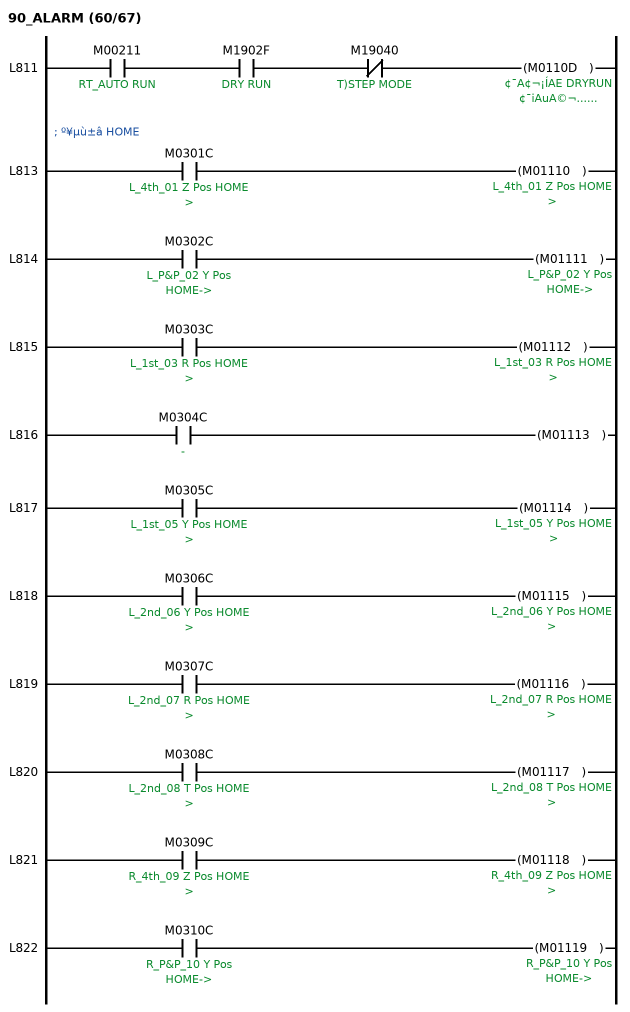
[picture p456: 90_ALARM rungs L811-L822]
; L811
LOAD      M00211	// RT_AUTO RUN
AND       M1902F	// DRY RUN
AND NOT   M19040	// T)STEP MODE
OUT       M0110D	// ¢¯A¢¬¡ÍAE DRYRUN ¢¯iAuA©¬......
// º¥µù±â HOME
; L813
LOAD      M0301C	// L_4th_01 Z Pos HOME >
OUT       M01110	// L_4th_01 Z Pos HOME >
; L814
LOAD      M0302C	// L_P&P_02 Y Pos HOME->
OUT       M01111	// L_P&P_02 Y Pos HOME->
; L815
LOAD      M0303C	// L_1st_03 R Pos HOME >
OUT       M01112	// L_1st_03 R Pos HOME >
; L816
LOAD      M0304C	// -
OUT       M01113
; L817
LOAD      M0305C	// L_1st_05 Y Pos HOME >
OUT       M01114	// L_1st_05 Y Pos HOME >
; L818
LOAD      M0306C	// L_2nd_06 Y Pos HOME >
OUT       M01115	// L_2nd_06 Y Pos HOME >
; L819
LOAD      M0307C	// L_2nd_07 R Pos HOME >
OUT       M01116	// L_2nd_07 R Pos HOME >
; L820
LOAD      M0308C	// L_2nd_08 T Pos HOME >
OUT       M01117	// L_2nd_08 T Pos HOME >
; L821
LOAD      M0309C	// R_4th_09 Z Pos HOME >
OUT       M01118	// R_4th_09 Z Pos HOME >
; L822
LOAD      M0310C	// R_P&P_10 Y Pos HOME->
OUT       M01119	// R_P&P_10 Y Pos HOME->

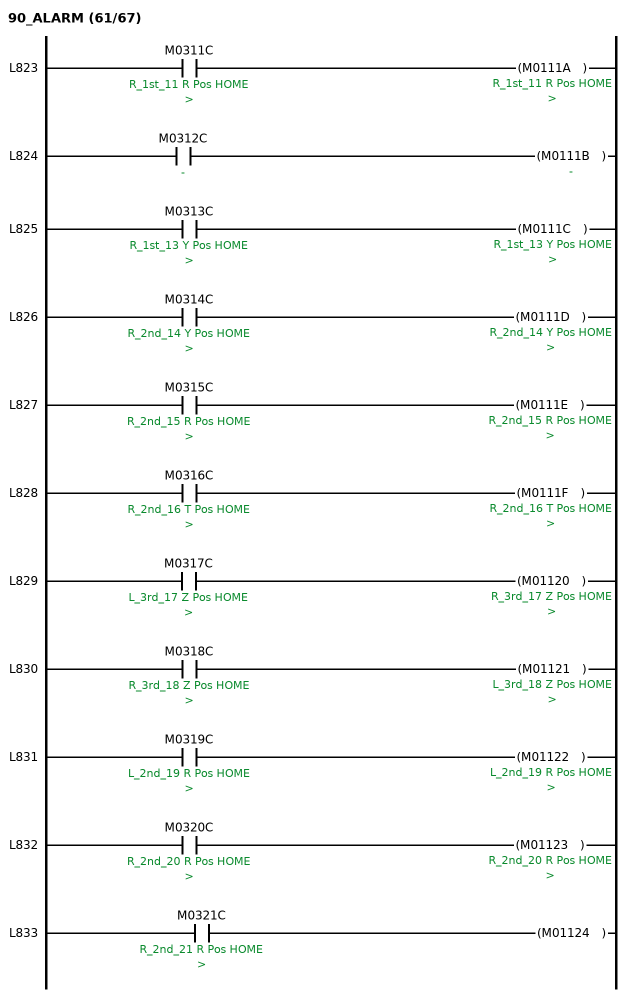
; L823
LOAD      M0311C	// R_1st_11 R Pos HOME >
OUT       M0111A	// R_1st_11 R Pos HOME >
; L824
LOAD      M0312C	// -
OUT       M0111B	// -
; L825
LOAD      M0313C	// R_1st_13 Y Pos HOME >
OUT       M0111C	// R_1st_13 Y Pos HOME >
; L826
LOAD      M0314C	// R_2nd_14 Y Pos HOME >
OUT       M0111D	// R_2nd_14 Y Pos HOME >
; L827
LOAD      M0315C	// R_2nd_15 R Pos HOME >
OUT       M0111E	// R_2nd_15 R Pos HOME >
; L828
LOAD      M0316C	// R_2nd_16 T Pos HOME >
OUT       M0111F	// R_2nd_16 T Pos HOME >
; L829
LOAD      M0317C	// L_3rd_17 Z Pos HOME >
OUT       M01120	// R_3rd_17 Z Pos HOME >
; L830
LOAD      M0318C	// R_3rd_18 Z Pos HOME >
OUT       M01121	// L_3rd_18 Z Pos HOME >
; L831
LOAD      M0319C	// L_2nd_19 R Pos HOME >
OUT       M01122	// L_2nd_19 R Pos HOME >
; L832
LOAD      M0320C	// R_2nd_20 R Pos HOME >
OUT       M01123	// R_2nd_20 R Pos HOME >
; L833
LOAD      M0321C	// R_2nd_21 R Pos HOME >
OUT       M01124

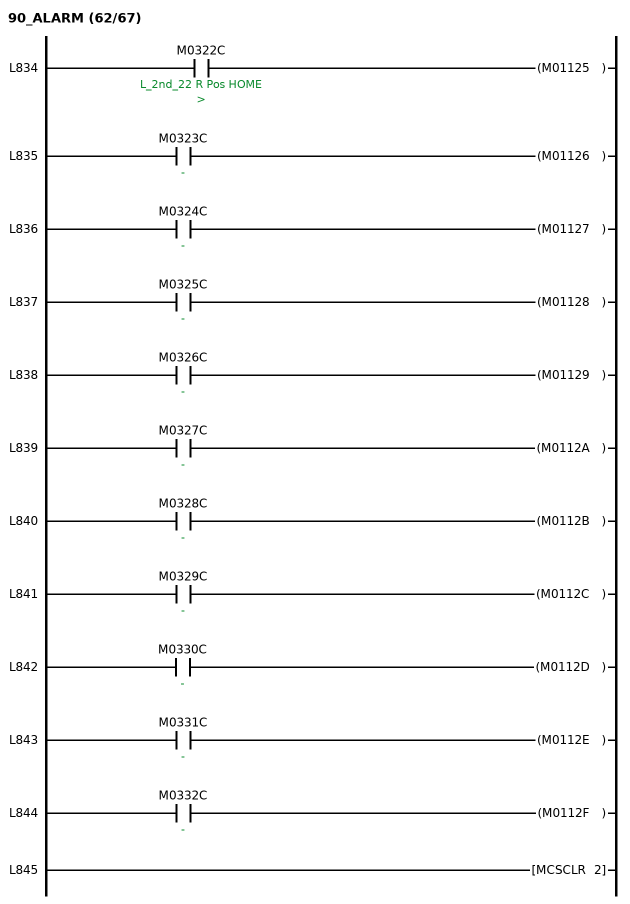
; L834
LOAD      M0322C	// L_2nd_22 R Pos HOME >
OUT       M01125
; L835
LOAD      M0323C	// -
OUT       M01126
; L836
LOAD      M0324C	// -
OUT       M01127
; L837
LOAD      M0325C	// -
OUT       M01128
; L838
LOAD      M0326C	// -
OUT       M01129
; L839
LOAD      M0327C	// -
OUT       M0112A
; L840
LOAD      M0328C	// -
OUT       M0112B
; L841
LOAD      M0329C	// -
OUT       M0112C
; L842
LOAD      M0330C	// -
OUT       M0112D
; L843
LOAD      M0331C	// -
OUT       M0112E
; L844
LOAD      M0332C	// -
OUT       M0112F
; L845
MCSCLR    2

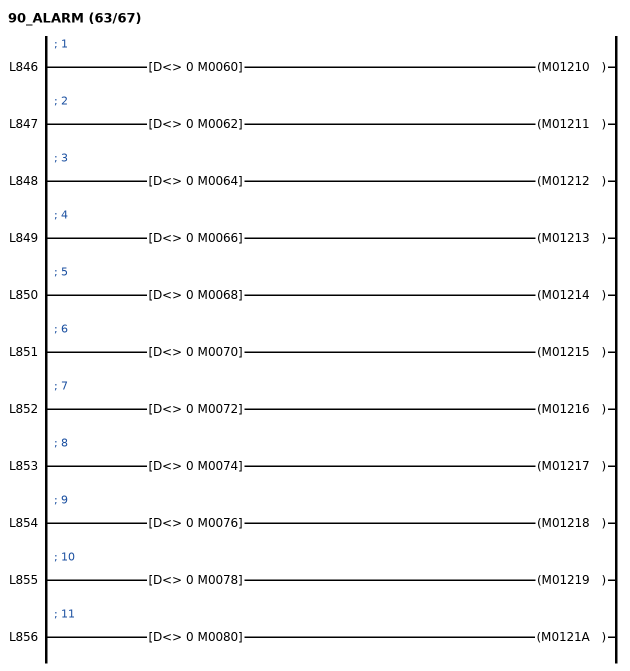
; L846
LOADD<>   0 M0060
OUT       M01210
// output comment: 1
; L847
LOADD<>   0 M0062
OUT       M01211
// output comment: 2
; L848
LOADD<>   0 M0064
OUT       M01212
// output comment: 3
; L849
LOADD<>   0 M0066
OUT       M01213
// output comment: 4
; L850
LOADD<>   0 M0068
OUT       M01214
// output comment: 5
; L851
LOADD<>   0 M0070
OUT       M01215
// output comment: 6
; L852
LOADD<>   0 M0072
OUT       M01216
// output comment: 7
; L853
LOADD<>   0 M0074
OUT       M01217
// output comment: 8
; L854
LOADD<>   0 M0076
OUT       M01218
// output comment: 9
; L855
LOADD<>   0 M0078
OUT       M01219
// output comment: 10
; L856
LOADD<>   0 M0080
OUT       M0121A
// output comment: 11

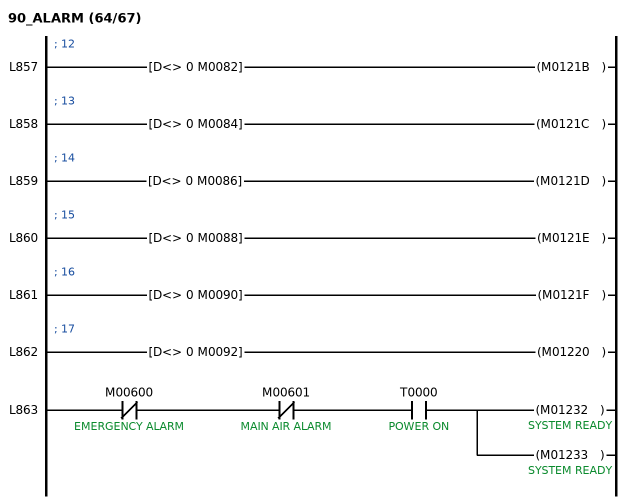
; L857
LOADD<>   0 M0082
OUT       M0121B
// output comment: 12
; L858
LOADD<>   0 M0084
OUT       M0121C
// output comment: 13
; L859
LOADD<>   0 M0086
OUT       M0121D
// output comment: 14
; L860
LOADD<>   0 M0088
OUT       M0121E
// output comment: 15
; L861
LOADD<>   0 M0090
OUT       M0121F
// output comment: 16
; L862
LOADD<>   0 M0092
OUT       M01220
// output comment: 17
; L863
LOAD NOT  M00600	// EMERGENCY ALARM
AND NOT   M00601	// MAIN AIR ALARM
AND       T0000	// POWER ON
OUT       M01232	// SYSTEM READY
OUT       M01233	// SYSTEM READY

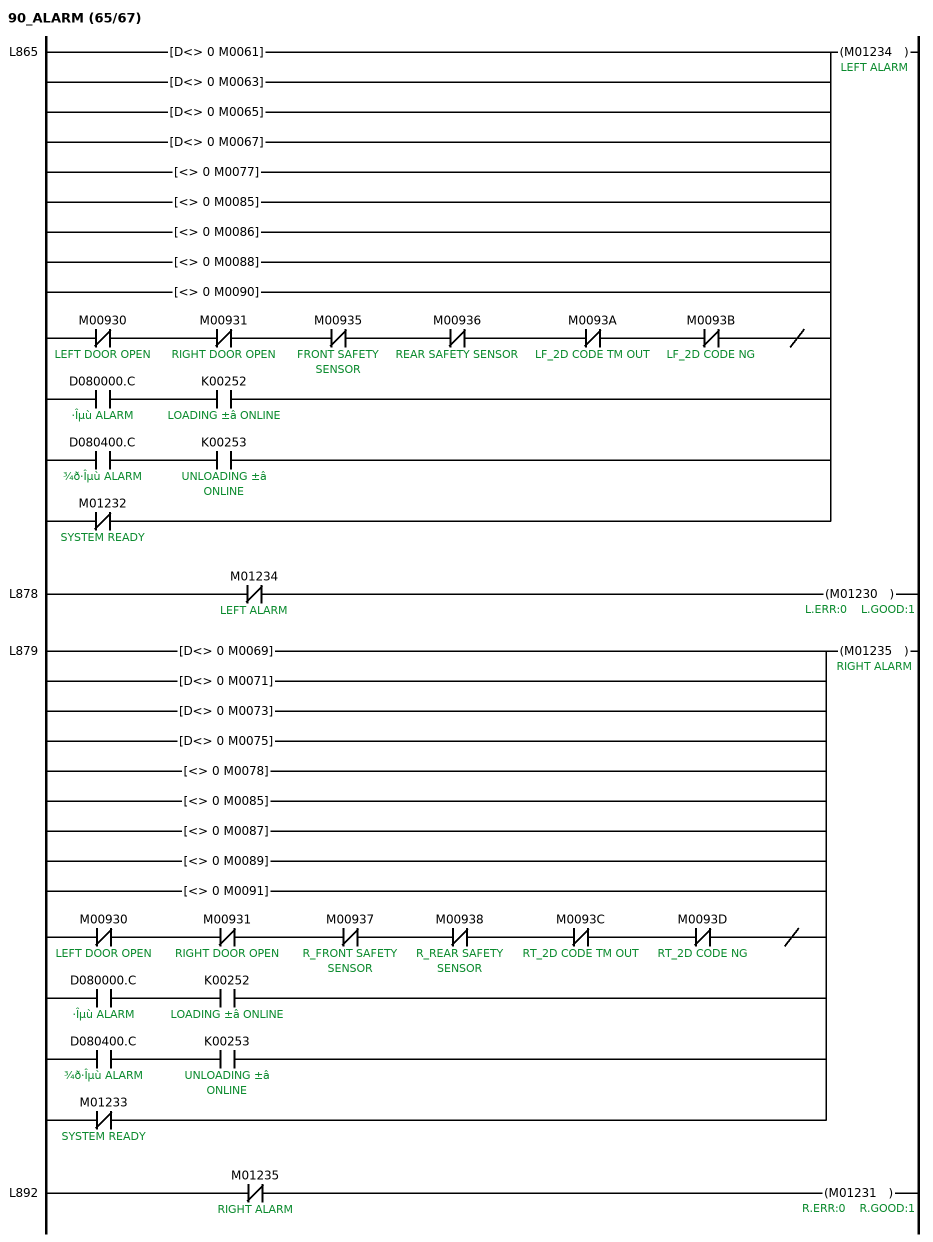
; L865
LOADD<>   0 M0061
ORD<>     0 M0063
ORD<>     0 M0065
ORD<>     0 M0067
OR<>      0 M0077
OR<>      0 M0085
OR<>      0 M0086
OR<>      0 M0088
OR<>      0 M0090
LOAD NOT  M00930	// LEFT DOOR OPEN
AND NOT   M00931	// RIGHT DOOR OPEN
AND NOT   M00935	// FRONT SAFETY SENSOR
AND NOT   M00936	// REAR SAFETY SENSOR
AND NOT   M0093A	// LF_2D CODE TM OUT
AND NOT   M0093B	// LF_2D CODE NG
NOT
OR LOAD
LOAD      D080000.C	// ·Îµù ALARM
AND       K00252	// LOADING ±â ONLINE
OR LOAD
LOAD      D080400.C	// ¾ð·Îµù ALARM
AND       K00253	// UNLOADING ±â ONLINE
OR LOAD
OR NOT    M01232	// SYSTEM READY
OUT       M01234	// LEFT ALARM
; L878
LOAD NOT  M01234	// LEFT ALARM
OUT       M01230	// L.ERR:0    L.GOOD:1
; L879
LOADD<>   0 M0069
ORD<>     0 M0071
ORD<>     0 M0073
ORD<>     0 M0075
OR<>      0 M0078
OR<>      0 M0085
OR<>      0 M0087
OR<>      0 M0089
OR<>      0 M0091
LOAD NOT  M00930	// LEFT DOOR OPEN
AND NOT   M00931	// RIGHT DOOR OPEN
AND NOT   M00937	// R_FRONT SAFETY SENSOR
AND NOT   M00938	// R_REAR SAFETY SENSOR
AND NOT   M0093C	// RT_2D CODE TM OUT
AND NOT   M0093D	// RT_2D CODE NG
NOT
OR LOAD
LOAD      D080000.C	// ·Îµù ALARM
AND       K00252	// LOADING ±â ONLINE
OR LOAD
LOAD      D080400.C	// ¾ð·Îµù ALARM
AND       K00253	// UNLOADING ±â ONLINE
OR LOAD
OR NOT    M01233	// SYSTEM READY
OUT       M01235	// RIGHT ALARM
; L892
LOAD NOT  M01235	// RIGHT ALARM
OUT       M01231	// R.ERR:0    R.GOOD:1

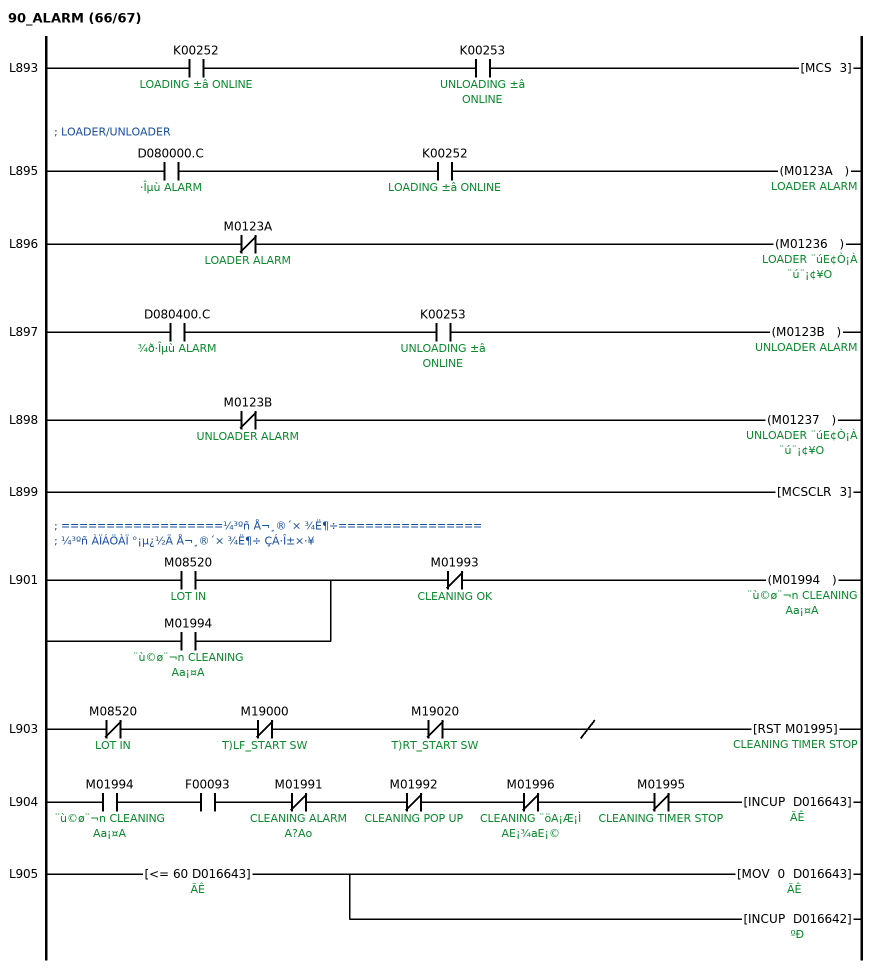
; L893
LOAD      K00252	// LOADING ±â ONLINE
AND       K00253	// UNLOADING ±â ONLINE
MCS       3
// LOADER/UNLOADER
; L895
LOAD      D080000.C	// ·Îµù ALARM
AND       K00252	// LOADING ±â ONLINE
OUT       M0123A	// LOADER ALARM
; L896
LOAD NOT  M0123A	// LOADER ALARM
OUT       M01236	// LOADER ¨úE¢Ò¡À ¨ú¨¡¢¥O
; L897
LOAD      D080400.C	// ¾ð·Îµù ALARM
AND       K00253	// UNLOADING ±â ONLINE
OUT       M0123B	// UNLOADER ALARM
; L898
LOAD NOT  M0123B	// UNLOADER ALARM
OUT       M01237	// UNLOADER ¨úE¢Ò¡À ¨ú¨¡¢¥O
; L899
MCSCLR    3
// ==================¼³ºñ Å¬¸®´× ¾Ë¶÷================
; L901
LOAD      M08520	// LOT IN
OR        M01994	// ¨ù©ø¨¬n CLEANING Aa¡¤A
AND NOT   M01993	// CLEANING OK
OUT       M01994	// ¨ù©ø¨¬n CLEANING Aa¡¤A
// output comment: ¼³ºñ ÀÏÁÖÀÏ °¡µ¿½Ã Å¬¸®´× ¾Ë¶÷ ÇÁ·Î±×·¥
; L903
LOAD NOT  M08520	// LOT IN
AND NOT   M19000	// T)LF_START SW
AND NOT   M19020	// T)RT_START SW
NOT
RST       M01995	// CLEANING TIMER STOP
; L904
LOAD      M01994	// ¨ù©ø¨¬n CLEANING Aa¡¤A
AND       F00093
AND NOT   M01991	// CLEANING ALARM A?Ao
AND NOT   M01992	// CLEANING POP UP
AND NOT   M01996	// CLEANING ¨öA¡Æ¡Ì AE¡¾aE¡©
AND NOT   M01995	// CLEANING TIMER STOP
INCUP     D016643	// ÃÊ
; L905
LOAD<=    60 D016643	// ÃÊ
MOV       0 D016643	// ÃÊ
INCUP     D016642	// ºÐ

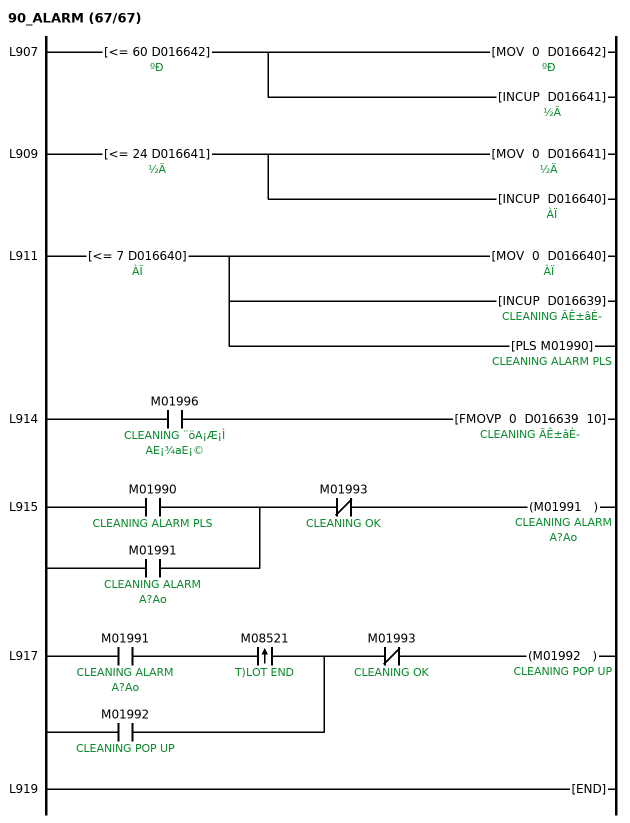
; L907
LOAD<=    60 D016642	// ºÐ
MOV       0 D016642	// ºÐ
INCUP     D016641	// ½Ã
; L909
LOAD<=    24 D016641	// ½Ã
MOV       0 D016641	// ½Ã
INCUP     D016640	// ÀÏ
; L911
LOAD<=    7 D016640	// ÀÏ
MOV       0 D016640	// ÀÏ
INCUP     D016639	// CLEANING ÃÊ±âÈ­
OUTP      M01990	// CLEANING ALARM PLS
; L914
LOAD      M01996	// CLEANING ¨öA¡Æ¡Ì AE¡¾aE¡©
FMOVP     0 D016639 10	// CLEANING ÃÊ±âÈ­
; L915
LOAD      M01990	// CLEANING ALARM PLS
OR        M01991	// CLEANING ALARM A?Ao
AND NOT   M01993	// CLEANING OK
OUT       M01991	// CLEANING ALARM A?Ao
; L917
LOAD      M01991	// CLEANING ALARM A?Ao
ANDP      M08521	// T)LOT END
OR        M01992	// CLEANING POP UP
AND NOT   M01993	// CLEANING OK
OUT       M01992	// CLEANING POP UP
; L919
END

PROGRAM 91_DEVICE_CHANGE (task: ½ºÄµ ÇÁ·Î±×·¥)

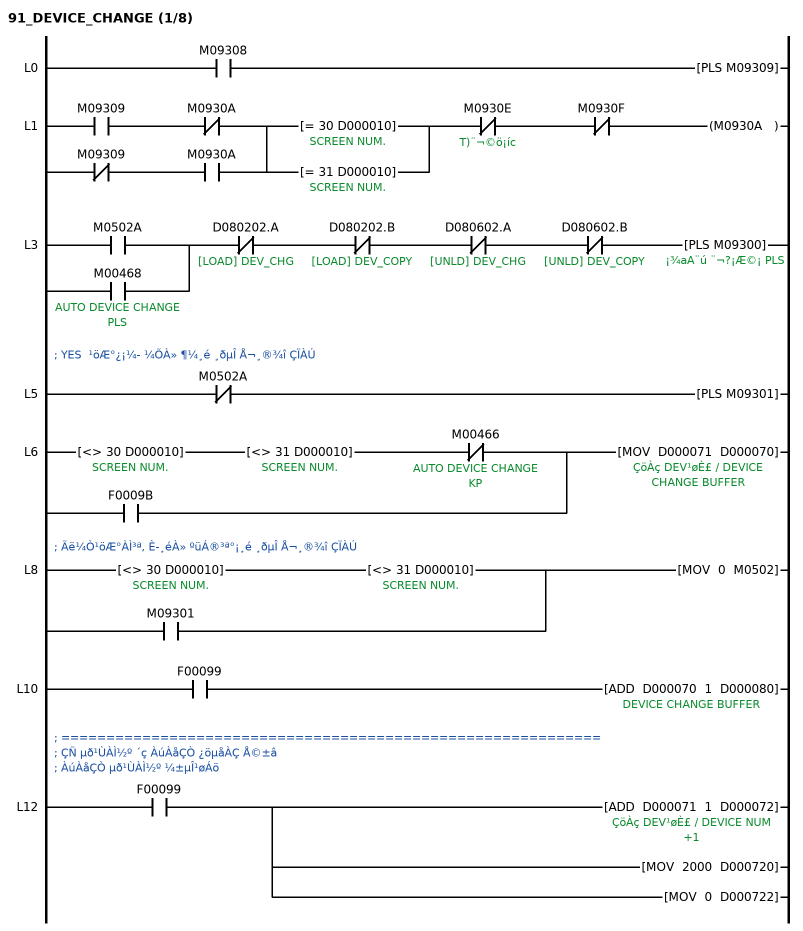
; L0
LOAD      M09308
OUTP      M09309
; L1
LOAD      M09309
AND NOT   M0930A
LOAD NOT  M09309
AND       M0930A
OR LOAD
LOAD=     30 D000010	// SCREEN NUM.
OR=       31 D000010	// SCREEN NUM.
AND LOAD
AND NOT   M0930E	// T)¨¬©ö¡íc
AND NOT   M0930F
OUT       M0930A
; L3
LOAD      M0502A
OR        M00468	// AUTO DEVICE CHANGE PLS
AND NOT   D080202.A	// [LOAD] DEV_CHG
AND NOT   D080202.B	// [LOAD] DEV_COPY
AND NOT   D080602.A	// [UNLD] DEV_CHG
AND NOT   D080602.B	// [UNLD] DEV_COPY
OUTP      M09300	// ¡¾aA¨ú ¨¬?¡Æ©¡ PLS
; L5
LOAD NOT  M0502A
OUTP      M09301
// output comment: YES  ¹öÆ°¿¡¼­ ¼ÕÀ» ¶¼¸é ¸ðµÎ Å¬¸®¾î ÇÏÀÚ
; L6
LOAD<>    30 D000010	// SCREEN NUM.
AND<>     31 D000010	// SCREEN NUM.
AND NOT   M00466	// AUTO DEVICE CHANGE KP
OR        F0009B
MOV       D000071 D000070	// ÇöÀç DEV¹øÈ£ / DEVICE CHANGE BUFFER
; L8
LOAD<>    30 D000010	// SCREEN NUM.
AND<>     31 D000010	// SCREEN NUM.
OR        M09301
MOV       0 M0502
// output comment: Ãë¼Ò¹öÆ°ÀÌ³ª, È­¸éÀ» ºüÁ®³ª°¡¸é ¸ðµÎ Å¬¸®¾î ÇÏÀÚ
; L10
LOAD      F00099
ADD       D000070 1 D000080	// DEVICE CHANGE BUFFER
// ============================================================
; L12
LOAD      F00099
ADD       D000071 1 D000072	// ÇöÀç DEV¹øÈ£ / DEVICE NUM +1
MOV       2000 D000720
MOV       0 D000722
// output comment: ÇÑ µð¹ÙÀÌ½º ´ç ÀúÀåÇÒ ¿öµåÀÇ Å©±â
// output comment: ÀúÀåÇÒ µð¹ÙÀÌ½º ¼±µÎ¹øÁö

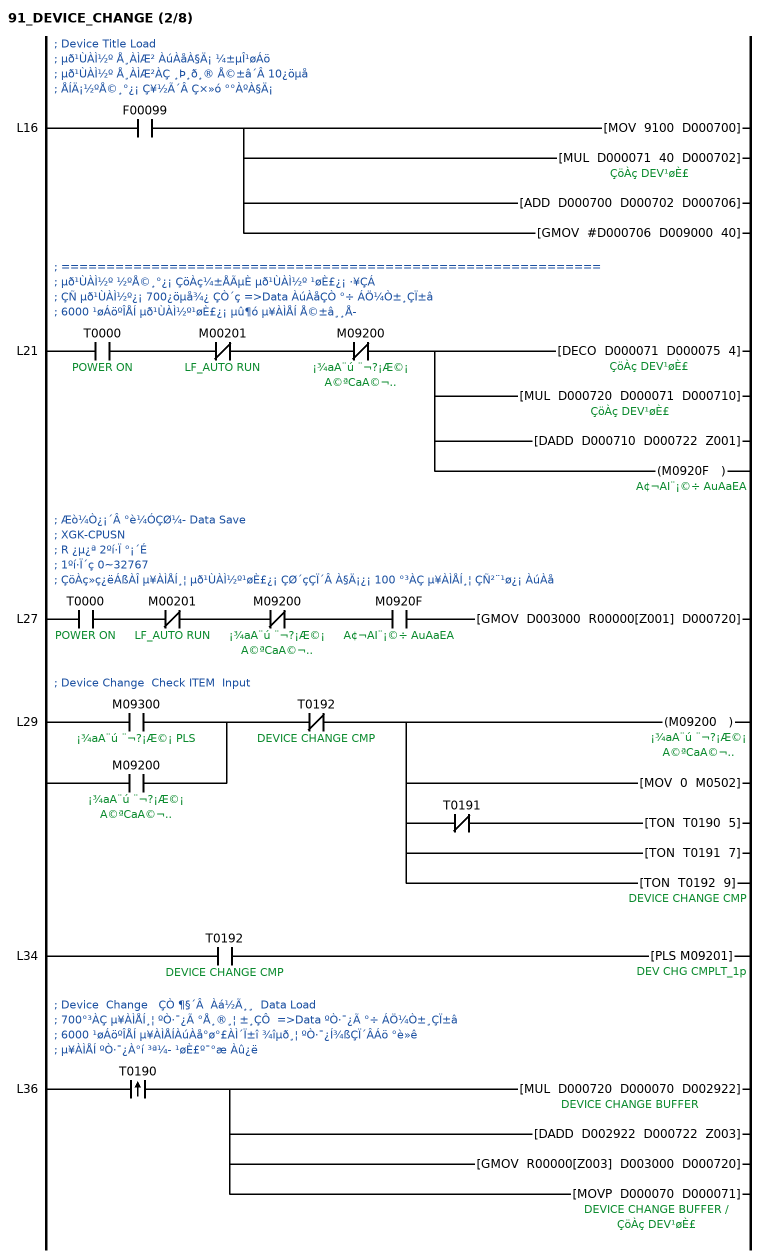
// Device Title Load
; L16
LOAD      F00099
MOV       9100 D000700
MUL       D000071 40 D000702	// ÇöÀç DEV¹øÈ£
ADD       D000700 D000702 D000706
GMOV      #D000706 D009000 40
// output comment: µð¹ÙÀÌ½º Å¸ÀÌÆ² ÀúÀåÀ§Ä¡ ¼±µÎ¹øÁö
// output comment: µð¹ÙÀÌ½º Å¸ÀÌÆ²ÀÇ ¸Þ¸ð¸® Å©±â´Â 10¿öµå
// output comment: ÅÍÄ¡½ºÅ©¸°¿¡ Ç¥½Ã´Â Ç×»ó °°ÀºÀ§Ä¡
// ============================================================
; L21
LOAD      T0000	// POWER ON
AND NOT   M00201	// LF_AUTO RUN
AND NOT   M09200	// ¡¾aA¨ú ¨¬?¡Æ©¡ A©ªCaA©¬..
DECO      D000071 D000075 4	// ÇöÀç DEV¹øÈ£
MUL       D000720 D000071 D000710	// ÇöÀç DEV¹øÈ£
DADD      D000710 D000722 Z001
OUT       M0920F	// A¢¬AI¨¡©÷ AuAaEA
// output comment: µð¹ÙÀÌ½º ½ºÅ©¸°¿¡ ÇöÀç¼±ÅÃµÈ µð¹ÙÀÌ½º ¹øÈ£¿¡ ·¥ÇÁ
// output comment: ÇÑ µð¹ÙÀÌ½º¿¡ 700¿öµå¾¿ ÇÒ´ç =>Data ÀúÀåÇÒ °÷ ÁÖ¼Ò±¸ÇÏ±â
// output comment: 6000 ¹øÁöºÎÅÍ µð¹ÙÀÌ½º¹øÈ£¿¡ µû¶ó µ¥ÀÌÅÍ Å©±â¸¸Å­
// Æò¼Ò¿¡´Â °è¼ÓÇØ¼­ Data Save
// XGK-CPUSN
// R ¿µ¿ª 2ºí·Ï °¡´É
// 1ºí·Ï´ç 0~32767
; L27
LOAD      T0000	// POWER ON
AND NOT   M00201	// LF_AUTO RUN
AND NOT   M09200	// ¡¾aA¨ú ¨¬?¡Æ©¡ A©ªCaA©¬..
AND       M0920F	// A¢¬AI¨¡©÷ AuAaEA
GMOV      D003000 R00000[Z001] D000720
// output comment: ÇöÀç»ç¿ëÁßÀÎ µ¥ÀÌÅÍ¸¦ µð¹ÙÀÌ½º¹øÈ£¿¡ ÇØ´çÇÏ´Â À§Ä¡¿¡ 100 °³ÀÇ µ¥ÀÌÅÍ¸¦ ÇÑ²¨¹ø¿¡ ÀúÀå
// Device Change  Check ITEM  Input
; L29
LOAD      M09300	// ¡¾aA¨ú ¨¬?¡Æ©¡ PLS
OR        M09200	// ¡¾aA¨ú ¨¬?¡Æ©¡ A©ªCaA©¬..
AND NOT   T0192	// DEVICE CHANGE CMP
OUT       M09200	// ¡¾aA¨ú ¨¬?¡Æ©¡ A©ªCaA©¬..
MOV       0 M0502
MPUSH
AND NOT   T0191
TON       T0190 5
MPOP
TON       T0191 7
TON       T0192 9	// DEVICE CHANGE CMP
; L34
LOAD      T0192	// DEVICE CHANGE CMP
OUTP      M09201	// DEV CHG CMPLT_1p
// Device  Change   ÇÒ ¶§´Â  Àá½Ã¸¸  Data Load
; L36
LOADP     T0190
MUL       D000720 D000070 D002922	// DEVICE CHANGE BUFFER
DADD      D002922 D000722 Z003
GMOV      R00000[Z003] D003000 D000720
MOVP      D000070 D000071	// DEVICE CHANGE BUFFER / ÇöÀç DEV¹øÈ£
// output comment: 700°³ÀÇ µ¥ÀÌÅÍ¸¦ ºÒ·¯¿Ã °Å¸®¸¦ ±¸ÇÔ  =>Data ºÒ·¯¿Ã °÷ ÁÖ¼Ò±¸ÇÏ±â
// output comment: 6000 ¹øÁöºÎÅÍ µ¥ÀÌÅÍÀúÀå°ø°£ÀÌ´Ï±î ¾îµð¸¦ ºÒ·¯¿Í¾ßÇÏ´ÂÁö °è»ê
// output comment: µ¥ÀÌÅÍ ºÒ·¯¿À°í ³ª¼­ ¹øÈ£º¯°æ Àû¿ë

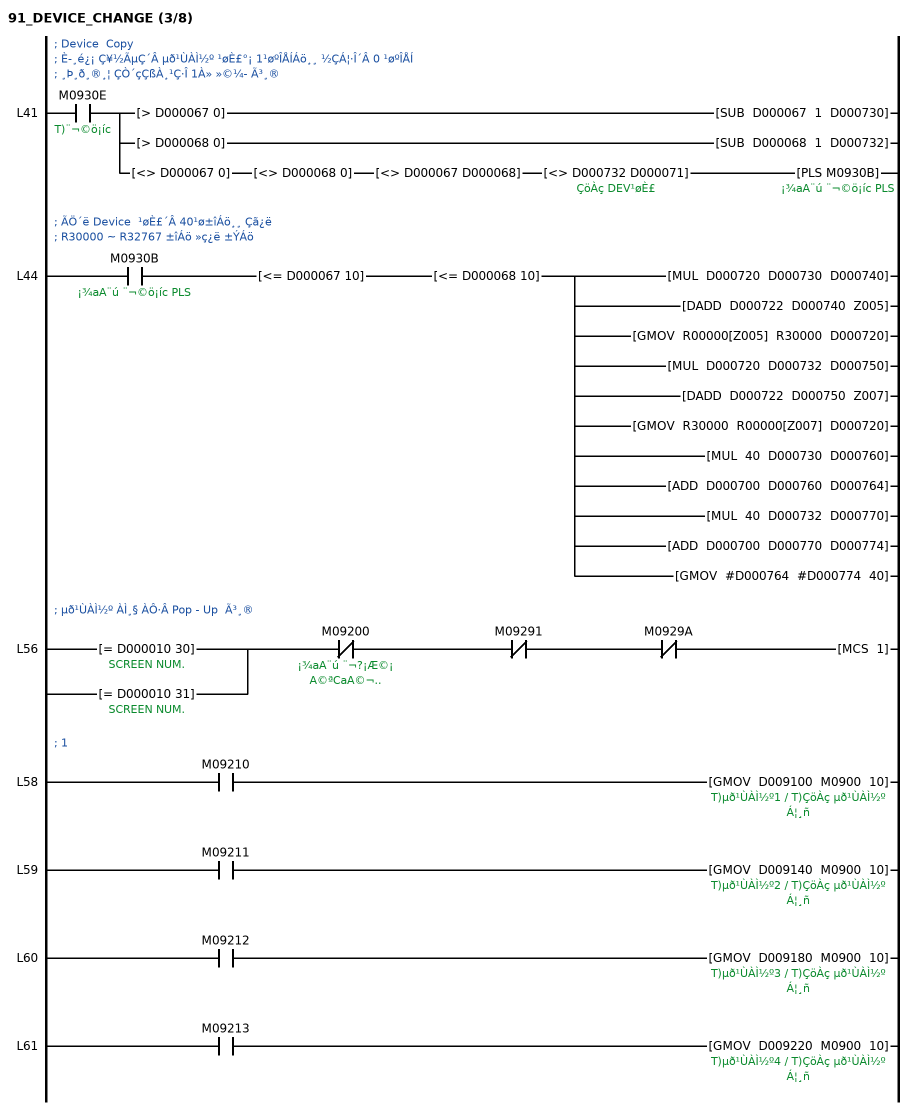
// Device  Copy
; L41
LOAD      M0930E	// T)¨¬©ö¡íc
MPUSH
AND>      D000067 0
SUB       D000067 1 D000730
MLOAD
AND>      D000068 0
SUB       D000068 1 D000732
MPOP
AND<>     D000067 0
AND<>     D000068 0
AND<>     D000067 D000068
AND<>     D000732 D000071	// ÇöÀç DEV¹øÈ£
OUTP      M0930B	// ¡¾aA¨ú ¨¬©ö¡íc PLS
// output comment: È­¸é¿¡ Ç¥½ÃµÇ´Â µð¹ÙÀÌ½º ¹øÈ£°¡ 1¹øºÎÅÍÁö¸¸ ½ÇÁ¦·Î´Â 0 ¹øºÎÅÍ
// output comment: ¸Þ¸ð¸®¸¦ ÇÒ´çÇßÀ¸¹Ç·Î 1À» »©¼­ Ã³¸®
; L44
LOAD      M0930B	// ¡¾aA¨ú ¨¬©ö¡íc PLS
AND<=     D000067 10
AND<=     D000068 10
MUL       D000720 D000730 D000740
DADD      D000722 D000740 Z005
GMOV      R00000[Z005] R30000 D000720
MUL       D000720 D000732 D000750
DADD      D000722 D000750 Z007
GMOV      R30000 R00000[Z007] D000720
MUL       40 D000730 D000760
ADD       D000700 D000760 D000764
MUL       40 D000732 D000770
ADD       D000700 D000770 D000774
GMOV      #D000764 #D000774 40
// output comment: ÃÖ´ë Device  ¹øÈ£´Â 40¹ø±îÁö¸¸ Çã¿ë
// output comment: R30000 ~ R32767 ±îÁö »ç¿ë ±ÝÁö
// µð¹ÙÀÌ½º ÀÌ¸§ ÀÔ·Â Pop - Up  Ã³¸®
; L56
LOAD=     D000010 30	// SCREEN NUM.
OR=       D000010 31	// SCREEN NUM.
AND NOT   M09200	// ¡¾aA¨ú ¨¬?¡Æ©¡ A©ªCaA©¬..
AND NOT   M09291
AND NOT   M0929A
MCS       1
; L58
LOAD      M09210
GMOV      D009100 M0900 10	// T)µð¹ÙÀÌ½º1 / T)ÇöÀç µð¹ÙÀÌ½º Á¦¸ñ
// output comment: 1
; L59
LOAD      M09211
GMOV      D009140 M0900 10	// T)µð¹ÙÀÌ½º2 / T)ÇöÀç µð¹ÙÀÌ½º Á¦¸ñ
; L60
LOAD      M09212
GMOV      D009180 M0900 10	// T)µð¹ÙÀÌ½º3 / T)ÇöÀç µð¹ÙÀÌ½º Á¦¸ñ
; L61
LOAD      M09213
GMOV      D009220 M0900 10	// T)µð¹ÙÀÌ½º4 / T)ÇöÀç µð¹ÙÀÌ½º Á¦¸ñ

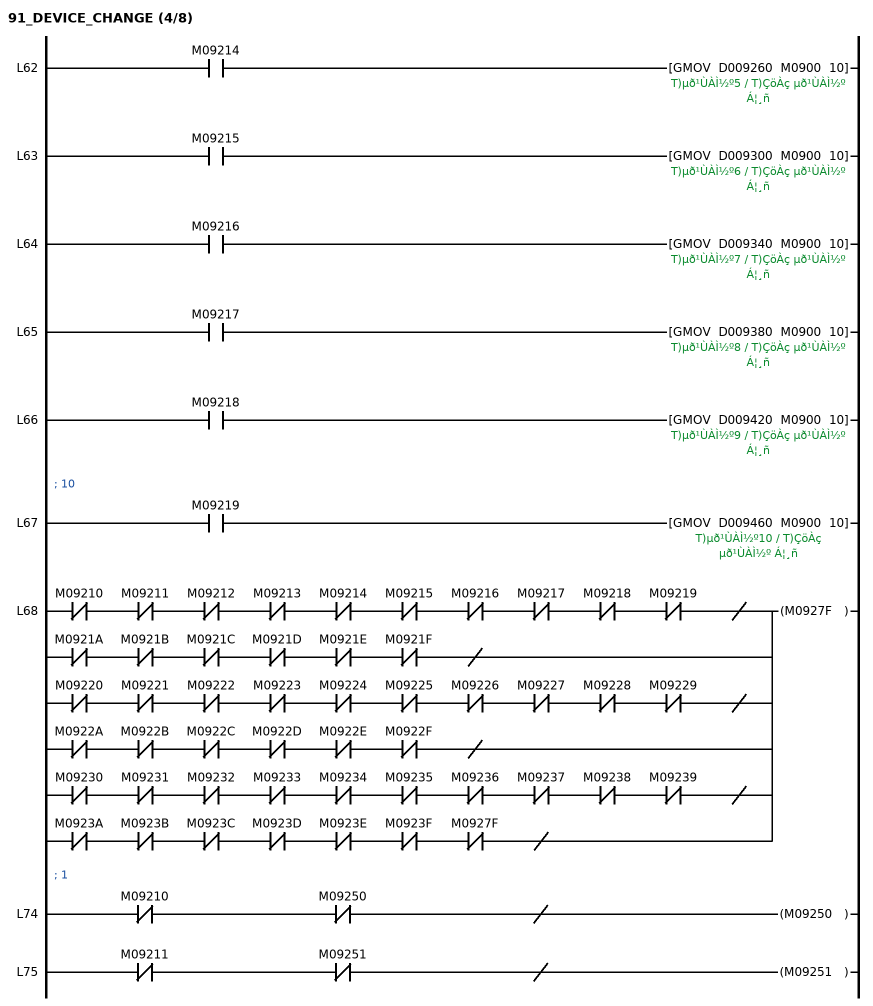
; L62
LOAD      M09214
GMOV      D009260 M0900 10	// T)µð¹ÙÀÌ½º5 / T)ÇöÀç µð¹ÙÀÌ½º Á¦¸ñ
; L63
LOAD      M09215
GMOV      D009300 M0900 10	// T)µð¹ÙÀÌ½º6 / T)ÇöÀç µð¹ÙÀÌ½º Á¦¸ñ
; L64
LOAD      M09216
GMOV      D009340 M0900 10	// T)µð¹ÙÀÌ½º7 / T)ÇöÀç µð¹ÙÀÌ½º Á¦¸ñ
; L65
LOAD      M09217
GMOV      D009380 M0900 10	// T)µð¹ÙÀÌ½º8 / T)ÇöÀç µð¹ÙÀÌ½º Á¦¸ñ
; L66
LOAD      M09218
GMOV      D009420 M0900 10	// T)µð¹ÙÀÌ½º9 / T)ÇöÀç µð¹ÙÀÌ½º Á¦¸ñ
; L67
LOAD      M09219
GMOV      D009460 M0900 10	// T)µð¹ÙÀÌ½º10 / T)ÇöÀç µð¹ÙÀÌ½º Á¦¸ñ
// output comment: 10
; L68
LOAD NOT  M09210
AND NOT   M09211
AND NOT   M09212
AND NOT   M09213
AND NOT   M09214
AND NOT   M09215
AND NOT   M09216
AND NOT   M09217
AND NOT   M09218
AND NOT   M09219
NOT
LOAD NOT  M0921A
AND NOT   M0921B
AND NOT   M0921C
AND NOT   M0921D
AND NOT   M0921E
AND NOT   M0921F
NOT
OR LOAD
LOAD NOT  M09220
AND NOT   M09221
AND NOT   M09222
AND NOT   M09223
AND NOT   M09224
AND NOT   M09225
AND NOT   M09226
AND NOT   M09227
AND NOT   M09228
AND NOT   M09229
NOT
OR LOAD
LOAD NOT  M0922A
AND NOT   M0922B
AND NOT   M0922C
AND NOT   M0922D
AND NOT   M0922E
AND NOT   M0922F
NOT
OR LOAD
LOAD NOT  M09230
AND NOT   M09231
AND NOT   M09232
AND NOT   M09233
AND NOT   M09234
AND NOT   M09235
AND NOT   M09236
AND NOT   M09237
AND NOT   M09238
AND NOT   M09239
NOT
OR LOAD
LOAD NOT  M0923A
AND NOT   M0923B
AND NOT   M0923C
AND NOT   M0923D
AND NOT   M0923E
AND NOT   M0923F
AND NOT   M0927F
NOT
OR LOAD
OUT       M0927F
; L74
LOAD NOT  M09210
AND NOT   M09250
NOT
OUT       M09250
// output comment: 1
; L75
LOAD NOT  M09211
AND NOT   M09251
NOT
OUT       M09251

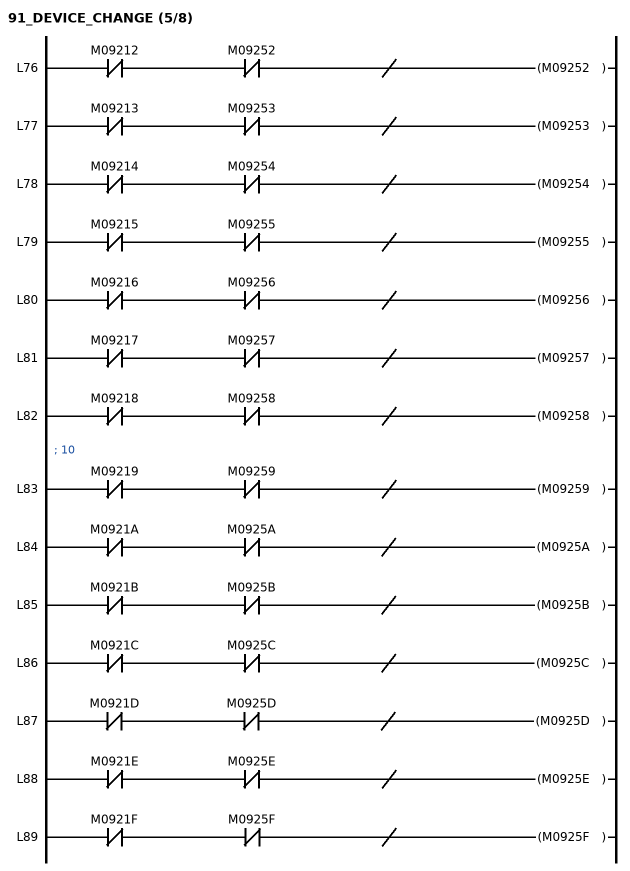
; L76
LOAD NOT  M09212
AND NOT   M09252
NOT
OUT       M09252
; L77
LOAD NOT  M09213
AND NOT   M09253
NOT
OUT       M09253
; L78
LOAD NOT  M09214
AND NOT   M09254
NOT
OUT       M09254
; L79
LOAD NOT  M09215
AND NOT   M09255
NOT
OUT       M09255
; L80
LOAD NOT  M09216
AND NOT   M09256
NOT
OUT       M09256
; L81
LOAD NOT  M09217
AND NOT   M09257
NOT
OUT       M09257
; L82
LOAD NOT  M09218
AND NOT   M09258
NOT
OUT       M09258
; L83
LOAD NOT  M09219
AND NOT   M09259
NOT
OUT       M09259
// output comment: 10
; L84
LOAD NOT  M0921A
AND NOT   M0925A
NOT
OUT       M0925A
; L85
LOAD NOT  M0921B
AND NOT   M0925B
NOT
OUT       M0925B
; L86
LOAD NOT  M0921C
AND NOT   M0925C
NOT
OUT       M0925C
; L87
LOAD NOT  M0921D
AND NOT   M0925D
NOT
OUT       M0925D
; L88
LOAD NOT  M0921E
AND NOT   M0925E
NOT
OUT       M0925E
; L89
LOAD NOT  M0921F
AND NOT   M0925F
NOT
OUT       M0925F

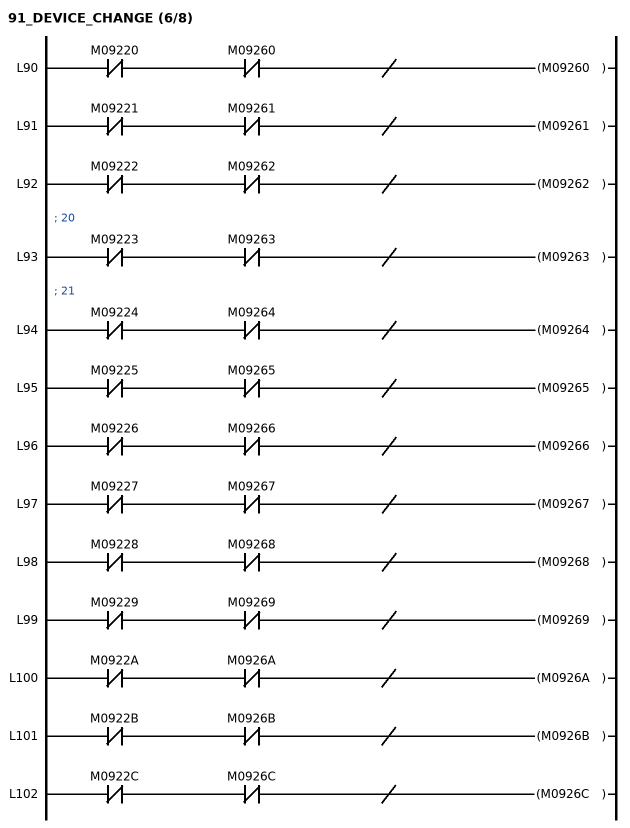
; L90
LOAD NOT  M09220
AND NOT   M09260
NOT
OUT       M09260
; L91
LOAD NOT  M09221
AND NOT   M09261
NOT
OUT       M09261
; L92
LOAD NOT  M09222
AND NOT   M09262
NOT
OUT       M09262
; L93
LOAD NOT  M09223
AND NOT   M09263
NOT
OUT       M09263
// output comment: 20
; L94
LOAD NOT  M09224
AND NOT   M09264
NOT
OUT       M09264
// output comment: 21
; L95
LOAD NOT  M09225
AND NOT   M09265
NOT
OUT       M09265
; L96
LOAD NOT  M09226
AND NOT   M09266
NOT
OUT       M09266
; L97
LOAD NOT  M09227
AND NOT   M09267
NOT
OUT       M09267
; L98
LOAD NOT  M09228
AND NOT   M09268
NOT
OUT       M09268
; L99
LOAD NOT  M09229
AND NOT   M09269
NOT
OUT       M09269
; L100
LOAD NOT  M0922A
AND NOT   M0926A
NOT
OUT       M0926A
; L101
LOAD NOT  M0922B
AND NOT   M0926B
NOT
OUT       M0926B
; L102
LOAD NOT  M0922C
AND NOT   M0926C
NOT
OUT       M0926C

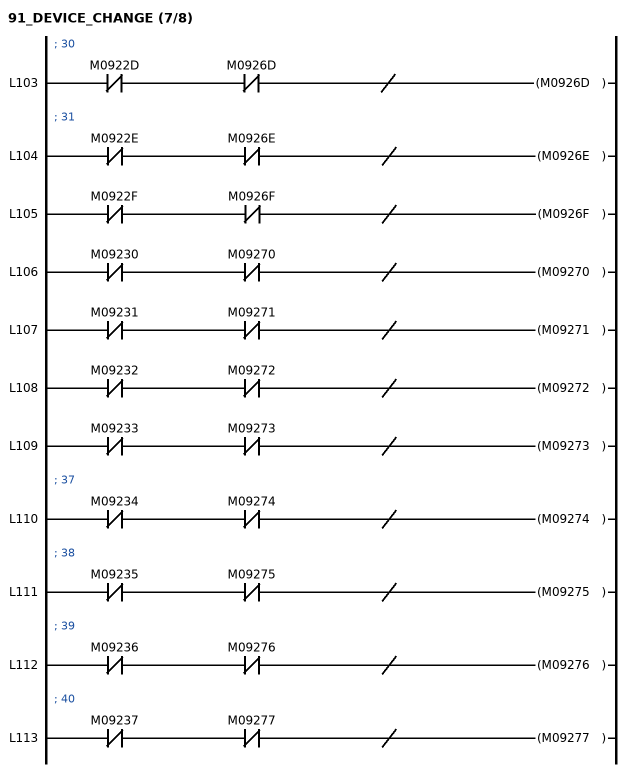
; L103
LOAD NOT  M0922D
AND NOT   M0926D
NOT
OUT       M0926D
// output comment: 30
; L104
LOAD NOT  M0922E
AND NOT   M0926E
NOT
OUT       M0926E
// output comment: 31
; L105
LOAD NOT  M0922F
AND NOT   M0926F
NOT
OUT       M0926F
; L106
LOAD NOT  M09230
AND NOT   M09270
NOT
OUT       M09270
; L107
LOAD NOT  M09231
AND NOT   M09271
NOT
OUT       M09271
; L108
LOAD NOT  M09232
AND NOT   M09272
NOT
OUT       M09272
; L109
LOAD NOT  M09233
AND NOT   M09273
NOT
OUT       M09273
; L110
LOAD NOT  M09234
AND NOT   M09274
NOT
OUT       M09274
// output comment: 37
; L111
LOAD NOT  M09235
AND NOT   M09275
NOT
OUT       M09275
// output comment: 38
; L112
LOAD NOT  M09236
AND NOT   M09276
NOT
OUT       M09276
// output comment: 39
; L113
LOAD NOT  M09237
AND NOT   M09277
NOT
OUT       M09277
// output comment: 40

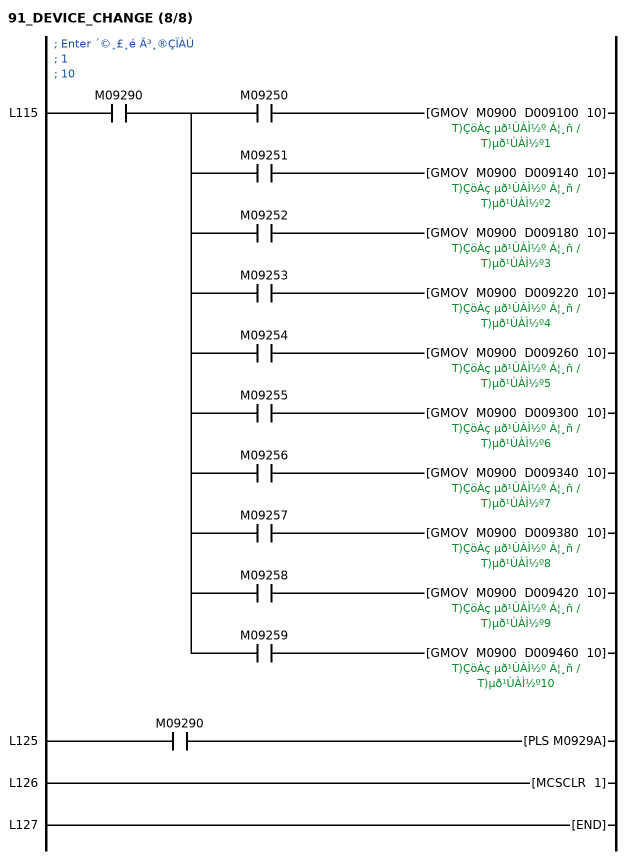
// Enter ´©¸£¸é Ã³¸®ÇÏÀÚ
; L115
LOAD      M09290
MPUSH
AND       M09250
GMOV      M0900 D009100 10	// T)ÇöÀç µð¹ÙÀÌ½º Á¦¸ñ / T)µð¹ÙÀÌ½º1
MLOAD
AND       M09251
GMOV      M0900 D009140 10	// T)ÇöÀç µð¹ÙÀÌ½º Á¦¸ñ / T)µð¹ÙÀÌ½º2
MLOAD
AND       M09252
GMOV      M0900 D009180 10	// T)ÇöÀç µð¹ÙÀÌ½º Á¦¸ñ / T)µð¹ÙÀÌ½º3
MLOAD
AND       M09253
GMOV      M0900 D009220 10	// T)ÇöÀç µð¹ÙÀÌ½º Á¦¸ñ / T)µð¹ÙÀÌ½º4
MLOAD
AND       M09254
GMOV      M0900 D009260 10	// T)ÇöÀç µð¹ÙÀÌ½º Á¦¸ñ / T)µð¹ÙÀÌ½º5
MLOAD
AND       M09255
GMOV      M0900 D009300 10	// T)ÇöÀç µð¹ÙÀÌ½º Á¦¸ñ / T)µð¹ÙÀÌ½º6
MLOAD
AND       M09256
GMOV      M0900 D009340 10	// T)ÇöÀç µð¹ÙÀÌ½º Á¦¸ñ / T)µð¹ÙÀÌ½º7
MLOAD
AND       M09257
GMOV      M0900 D009380 10	// T)ÇöÀç µð¹ÙÀÌ½º Á¦¸ñ / T)µð¹ÙÀÌ½º8
MLOAD
AND       M09258
GMOV      M0900 D009420 10	// T)ÇöÀç µð¹ÙÀÌ½º Á¦¸ñ / T)µð¹ÙÀÌ½º9
MPOP
AND       M09259
GMOV      M0900 D009460 10	// T)ÇöÀç µð¹ÙÀÌ½º Á¦¸ñ / T)µð¹ÙÀÌ½º10
// output comment: 1
// output comment: 10
; L125
LOAD      M09290
OUTP      M0929A
; L126
MCSCLR    1
; L127
END

PROGRAM 92_ALARM_SCR (task: ½ºÄµ ÇÁ·Î±×·¥)

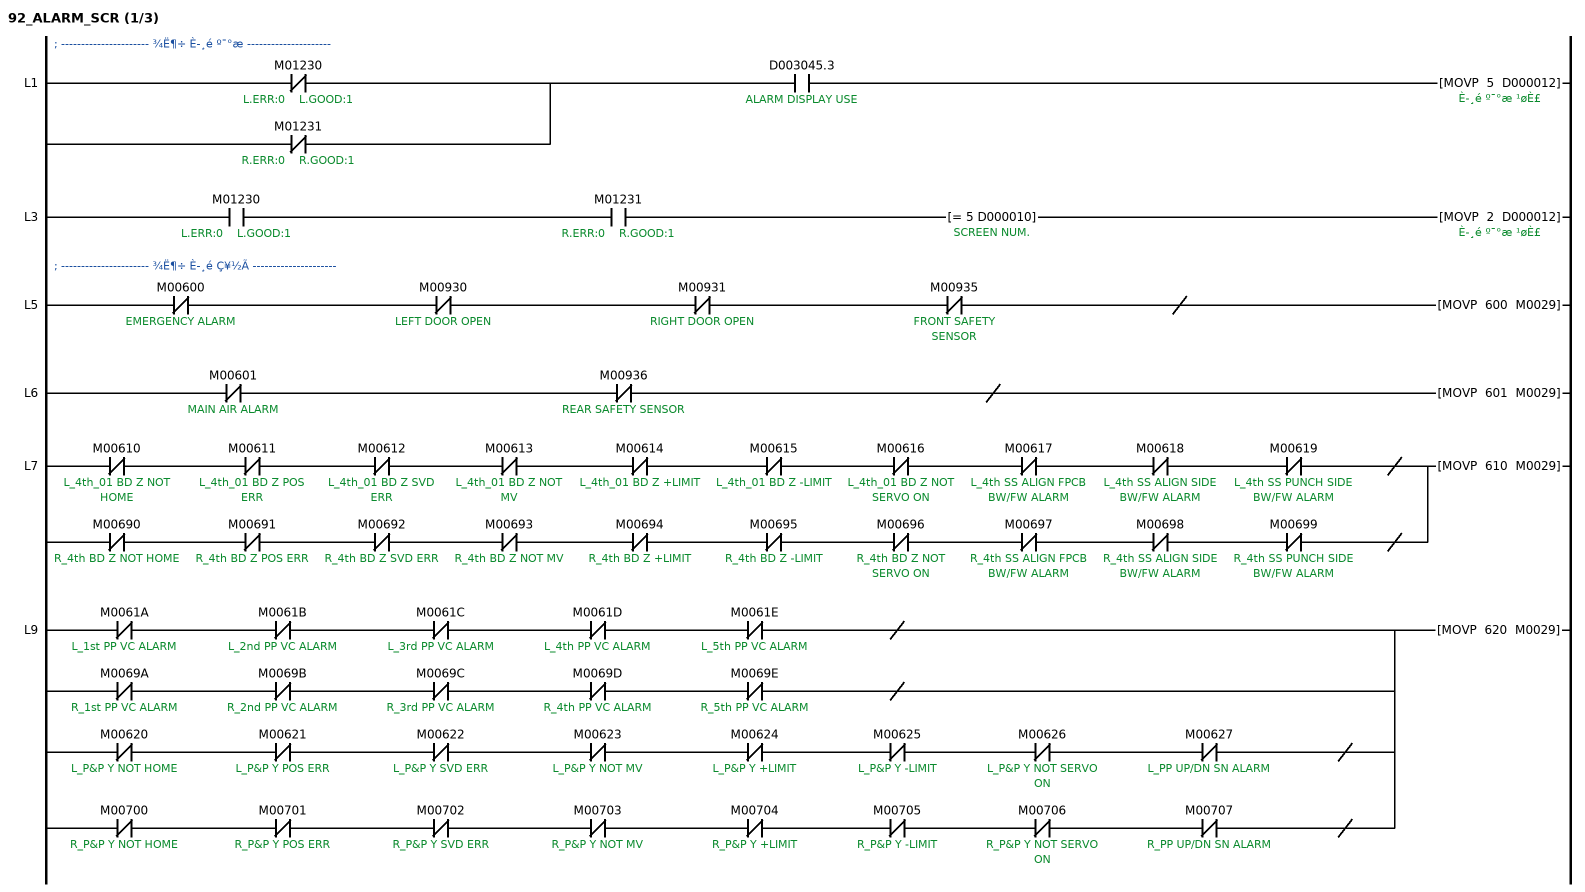
// ---------------------- ¾Ë¶÷ È­¸é º¯°æ ---------------------
; L1
LOAD NOT  M01230	// L.ERR:0    L.GOOD:1
OR NOT    M01231	// R.ERR:0    R.GOOD:1
AND       D003045.3	// ALARM DISPLAY USE
MOVP      5 D000012	// È­¸é º¯°æ ¹øÈ£
; L3
LOAD      M01230	// L.ERR:0    L.GOOD:1
AND       M01231	// R.ERR:0    R.GOOD:1
AND=      5 D000010	// SCREEN NUM.
MOVP      2 D000012	// È­¸é º¯°æ ¹øÈ£
// ---------------------- ¾Ë¶÷ È­¸é Ç¥½Ã ---------------------
; L5
LOAD NOT  M00600	// EMERGENCY ALARM
AND NOT   M00930	// LEFT DOOR OPEN
AND NOT   M00931	// RIGHT DOOR OPEN
AND NOT   M00935	// FRONT SAFETY SENSOR
NOT
MOVP      600 M0029
; L6
LOAD NOT  M00601	// MAIN AIR ALARM
AND NOT   M00936	// REAR SAFETY SENSOR
NOT
MOVP      601 M0029
; L7
LOAD NOT  M00610	// L_4th_01 BD Z NOT HOME
AND NOT   M00611	// L_4th_01 BD Z POS ERR
AND NOT   M00612	// L_4th_01 BD Z SVD ERR
AND NOT   M00613	// L_4th_01 BD Z NOT MV
AND NOT   M00614	// L_4th_01 BD Z +LIMIT
AND NOT   M00615	// L_4th_01 BD Z -LIMIT
AND NOT   M00616	// L_4th_01 BD Z NOT SERVO ON
AND NOT   M00617	// L_4th SS ALIGN FPCB BW/FW ALARM
AND NOT   M00618	// L_4th SS ALIGN SIDE BW/FW ALARM
AND NOT   M00619	// L_4th SS PUNCH SIDE BW/FW ALARM
NOT
LOAD NOT  M00690	// R_4th BD Z NOT HOME
AND NOT   M00691	// R_4th BD Z POS ERR
AND NOT   M00692	// R_4th BD Z SVD ERR
AND NOT   M00693	// R_4th BD Z NOT MV
AND NOT   M00694	// R_4th BD Z +LIMIT
AND NOT   M00695	// R_4th BD Z -LIMIT
AND NOT   M00696	// R_4th BD Z NOT SERVO ON
AND NOT   M00697	// R_4th SS ALIGN FPCB BW/FW ALARM
AND NOT   M00698	// R_4th SS ALIGN SIDE BW/FW ALARM
AND NOT   M00699	// R_4th SS PUNCH SIDE BW/FW ALARM
NOT
OR LOAD
MOVP      610 M0029
; L9
LOAD NOT  M0061A	// L_1st PP VC ALARM
AND NOT   M0061B	// L_2nd PP VC ALARM
AND NOT   M0061C	// L_3rd PP VC ALARM
AND NOT   M0061D	// L_4th PP VC ALARM
AND NOT   M0061E	// L_5th PP VC ALARM
NOT
LOAD NOT  M0069A	// R_1st PP VC ALARM
AND NOT   M0069B	// R_2nd PP VC ALARM
AND NOT   M0069C	// R_3rd PP VC ALARM
AND NOT   M0069D	// R_4th PP VC ALARM
AND NOT   M0069E	// R_5th PP VC ALARM
NOT
OR LOAD
LOAD NOT  M00620	// L_P&P Y NOT HOME
AND NOT   M00621	// L_P&P Y POS ERR
AND NOT   M00622	// L_P&P Y SVD ERR
AND NOT   M00623	// L_P&P Y NOT MV
AND NOT   M00624	// L_P&P Y +LIMIT
AND NOT   M00625	// L_P&P Y -LIMIT
AND NOT   M00626	// L_P&P Y NOT SERVO ON
AND NOT   M00627	// L_PP UP/DN SN ALARM
NOT
OR LOAD
LOAD NOT  M00700	// R_P&P Y NOT HOME
AND NOT   M00701	// R_P&P Y POS ERR
AND NOT   M00702	// R_P&P Y SVD ERR
AND NOT   M00703	// R_P&P Y NOT MV
AND NOT   M00704	// R_P&P Y +LIMIT
AND NOT   M00705	// R_P&P Y -LIMIT
AND NOT   M00706	// R_P&P Y NOT SERVO ON
AND NOT   M00707	// R_PP UP/DN SN ALARM
NOT
OR LOAD
MOVP      620 M0029

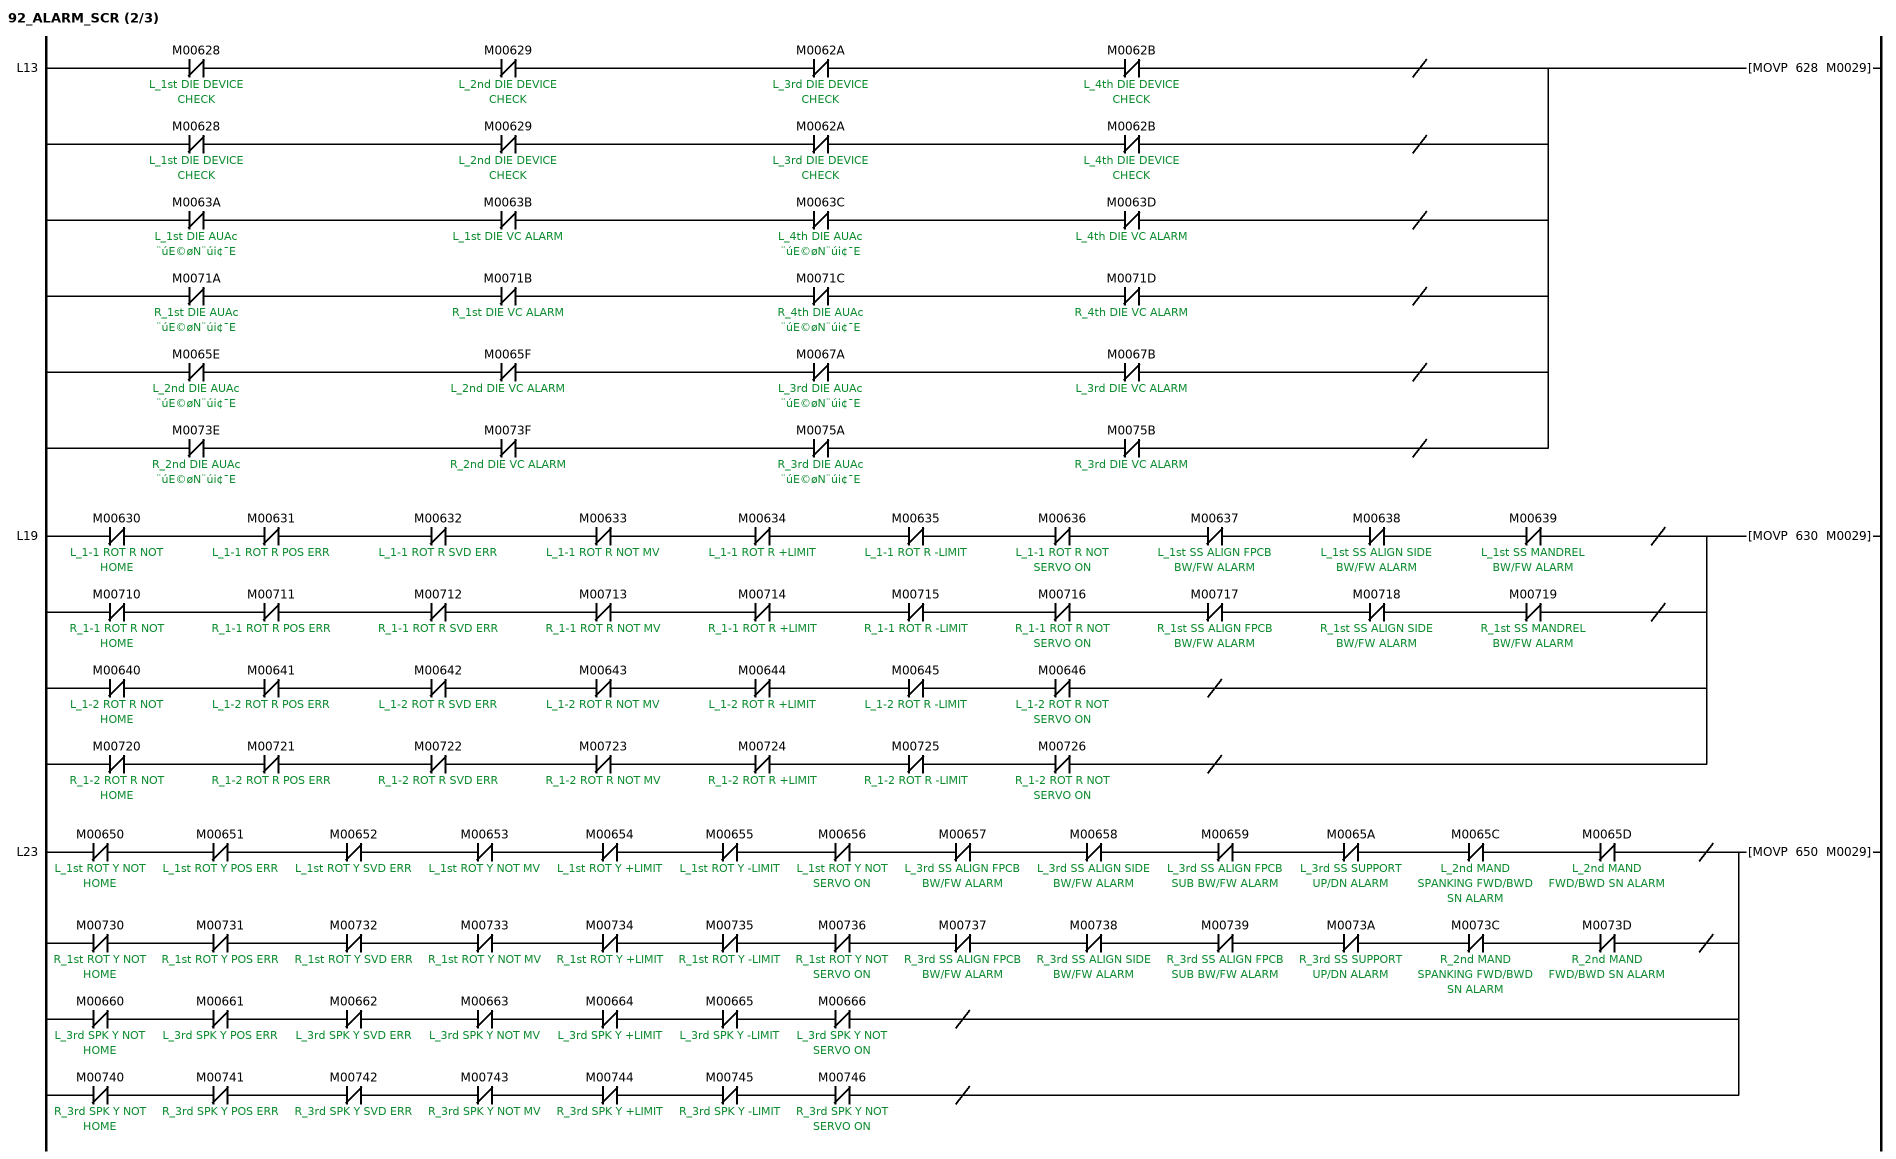
; L13
LOAD NOT  M00628	// L_1st DIE DEVICE CHECK
AND NOT   M00629	// L_2nd DIE DEVICE CHECK
AND NOT   M0062A	// L_3rd DIE DEVICE CHECK
AND NOT   M0062B	// L_4th DIE DEVICE CHECK
NOT
LOAD NOT  M00628	// L_1st DIE DEVICE CHECK
AND NOT   M00629	// L_2nd DIE DEVICE CHECK
AND NOT   M0062A	// L_3rd DIE DEVICE CHECK
AND NOT   M0062B	// L_4th DIE DEVICE CHECK
NOT
OR LOAD
LOAD NOT  M0063A	// L_1st DIE AUAc ¨úE©øN¨úi¢¯E
AND NOT   M0063B	// L_1st DIE VC ALARM
AND NOT   M0063C	// L_4th DIE AUAc ¨úE©øN¨úi¢¯E
AND NOT   M0063D	// L_4th DIE VC ALARM
NOT
OR LOAD
LOAD NOT  M0071A	// R_1st DIE AUAc ¨úE©øN¨úi¢¯E
AND NOT   M0071B	// R_1st DIE VC ALARM
AND NOT   M0071C	// R_4th DIE AUAc ¨úE©øN¨úi¢¯E
AND NOT   M0071D	// R_4th DIE VC ALARM
NOT
OR LOAD
LOAD NOT  M0065E	// L_2nd DIE AUAc ¨úE©øN¨úi¢¯E
AND NOT   M0065F	// L_2nd DIE VC ALARM
AND NOT   M0067A	// L_3rd DIE AUAc ¨úE©øN¨úi¢¯E
AND NOT   M0067B	// L_3rd DIE VC ALARM
NOT
OR LOAD
LOAD NOT  M0073E	// R_2nd DIE AUAc ¨úE©øN¨úi¢¯E
AND NOT   M0073F	// R_2nd DIE VC ALARM
AND NOT   M0075A	// R_3rd DIE AUAc ¨úE©øN¨úi¢¯E
AND NOT   M0075B	// R_3rd DIE VC ALARM
NOT
OR LOAD
MOVP      628 M0029
; L19
LOAD NOT  M00630	// L_1-1 ROT R NOT HOME
AND NOT   M00631	// L_1-1 ROT R POS ERR
AND NOT   M00632	// L_1-1 ROT R SVD ERR
AND NOT   M00633	// L_1-1 ROT R NOT MV
AND NOT   M00634	// L_1-1 ROT R +LIMIT
AND NOT   M00635	// L_1-1 ROT R -LIMIT
AND NOT   M00636	// L_1-1 ROT R NOT SERVO ON
AND NOT   M00637	// L_1st SS ALIGN FPCB BW/FW ALARM
AND NOT   M00638	// L_1st SS ALIGN SIDE BW/FW ALARM
AND NOT   M00639	// L_1st SS MANDREL BW/FW ALARM
NOT
LOAD NOT  M00710	// R_1-1 ROT R NOT HOME
AND NOT   M00711	// R_1-1 ROT R POS ERR
AND NOT   M00712	// R_1-1 ROT R SVD ERR
AND NOT   M00713	// R_1-1 ROT R NOT MV
AND NOT   M00714	// R_1-1 ROT R +LIMIT
AND NOT   M00715	// R_1-1 ROT R -LIMIT
AND NOT   M00716	// R_1-1 ROT R NOT SERVO ON
AND NOT   M00717	// R_1st SS ALIGN FPCB BW/FW ALARM
AND NOT   M00718	// R_1st SS ALIGN SIDE BW/FW ALARM
AND NOT   M00719	// R_1st SS MANDREL BW/FW ALARM
NOT
OR LOAD
LOAD NOT  M00640	// L_1-2 ROT R NOT HOME
AND NOT   M00641	// L_1-2 ROT R POS ERR
AND NOT   M00642	// L_1-2 ROT R SVD ERR
AND NOT   M00643	// L_1-2 ROT R NOT MV
AND NOT   M00644	// L_1-2 ROT R +LIMIT
AND NOT   M00645	// L_1-2 ROT R -LIMIT
AND NOT   M00646	// L_1-2 ROT R NOT SERVO ON
NOT
OR LOAD
LOAD NOT  M00720	// R_1-2 ROT R NOT HOME
AND NOT   M00721	// R_1-2 ROT R POS ERR
AND NOT   M00722	// R_1-2 ROT R SVD ERR
AND NOT   M00723	// R_1-2 ROT R NOT MV
AND NOT   M00724	// R_1-2 ROT R +LIMIT
AND NOT   M00725	// R_1-2 ROT R -LIMIT
AND NOT   M00726	// R_1-2 ROT R NOT SERVO ON
NOT
OR LOAD
MOVP      630 M0029
; L23
LOAD NOT  M00650	// L_1st ROT Y NOT HOME
AND NOT   M00651	// L_1st ROT Y POS ERR
AND NOT   M00652	// L_1st ROT Y SVD ERR
AND NOT   M00653	// L_1st ROT Y NOT MV
AND NOT   M00654	// L_1st ROT Y +LIMIT
AND NOT   M00655	// L_1st ROT Y -LIMIT
AND NOT   M00656	// L_1st ROT Y NOT SERVO ON
AND NOT   M00657	// L_3rd SS ALIGN FPCB BW/FW ALARM
AND NOT   M00658	// L_3rd SS ALIGN SIDE BW/FW ALARM
AND NOT   M00659	// L_3rd SS ALIGN FPCB SUB BW/FW ALARM
AND NOT   M0065A	// L_3rd SS SUPPORT UP/DN ALARM
AND NOT   M0065C	// L_2nd MAND SPANKING FWD/BWD SN ALARM
AND NOT   M0065D	// L_2nd MAND FWD/BWD SN ALARM
NOT
LOAD NOT  M00730	// R_1st ROT Y NOT HOME
AND NOT   M00731	// R_1st ROT Y POS ERR
AND NOT   M00732	// R_1st ROT Y SVD ERR
AND NOT   M00733	// R_1st ROT Y NOT MV
AND NOT   M00734	// R_1st ROT Y +LIMIT
AND NOT   M00735	// R_1st ROT Y -LIMIT
AND NOT   M00736	// R_1st ROT Y NOT SERVO ON
AND NOT   M00737	// R_3rd SS ALIGN FPCB BW/FW ALARM
AND NOT   M00738	// R_3rd SS ALIGN SIDE BW/FW ALARM
AND NOT   M00739	// R_3rd SS ALIGN FPCB SUB BW/FW ALARM
AND NOT   M0073A	// R_3rd SS SUPPORT UP/DN ALARM
AND NOT   M0073C	// R_2nd MAND SPANKING FWD/BWD SN ALARM
AND NOT   M0073D	// R_2nd MAND FWD/BWD SN ALARM
NOT
OR LOAD
LOAD NOT  M00660	// L_3rd SPK Y NOT HOME
AND NOT   M00661	// L_3rd SPK Y POS ERR
AND NOT   M00662	// L_3rd SPK Y SVD ERR
AND NOT   M00663	// L_3rd SPK Y NOT MV
AND NOT   M00664	// L_3rd SPK Y +LIMIT
AND NOT   M00665	// L_3rd SPK Y -LIMIT
AND NOT   M00666	// L_3rd SPK Y NOT SERVO ON
NOT
OR LOAD
LOAD NOT  M00740	// R_3rd SPK Y NOT HOME
AND NOT   M00741	// R_3rd SPK Y POS ERR
AND NOT   M00742	// R_3rd SPK Y SVD ERR
AND NOT   M00743	// R_3rd SPK Y NOT MV
AND NOT   M00744	// R_3rd SPK Y +LIMIT
AND NOT   M00745	// R_3rd SPK Y -LIMIT
AND NOT   M00746	// R_3rd SPK Y NOT SERVO ON
NOT
OR LOAD
MOVP      650 M0029

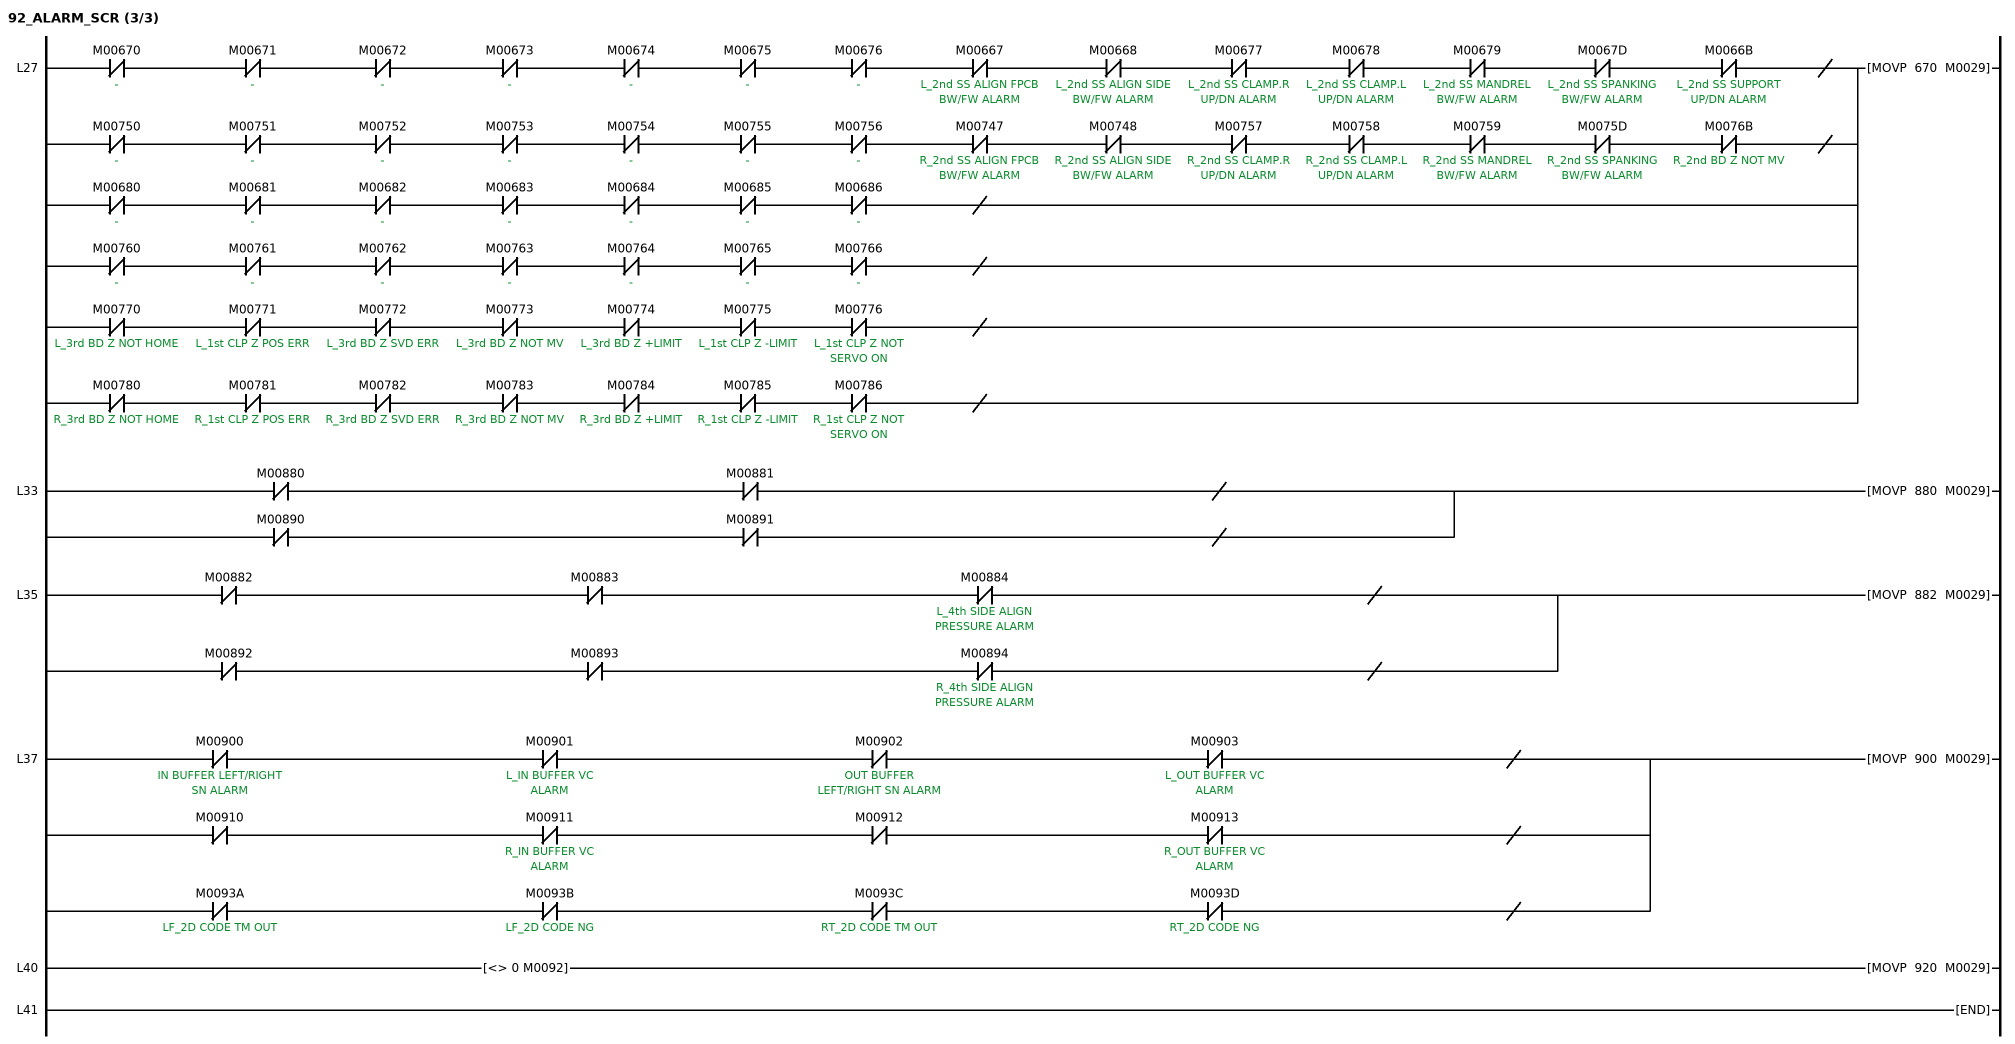
; L27
LOAD NOT  M00670	// -
AND NOT   M00671	// -
AND NOT   M00672	// -
AND NOT   M00673	// -
AND NOT   M00674	// -
AND NOT   M00675	// -
AND NOT   M00676	// -
AND NOT   M00667	// L_2nd SS ALIGN FPCB BW/FW ALARM
AND NOT   M00668	// L_2nd SS ALIGN SIDE BW/FW ALARM
AND NOT   M00677	// L_2nd SS CLAMP.R UP/DN ALARM
AND NOT   M00678	// L_2nd SS CLAMP.L UP/DN ALARM
AND NOT   M00679	// L_2nd SS MANDREL BW/FW ALARM
AND NOT   M0067D	// L_2nd SS SPANKING BW/FW ALARM
AND NOT   M0066B	// L_2nd SS SUPPORT UP/DN ALARM
NOT
LOAD NOT  M00750	// -
AND NOT   M00751	// -
AND NOT   M00752	// -
AND NOT   M00753	// -
AND NOT   M00754	// -
AND NOT   M00755	// -
AND NOT   M00756	// -
AND NOT   M00747	// R_2nd SS ALIGN FPCB BW/FW ALARM
AND NOT   M00748	// R_2nd SS ALIGN SIDE BW/FW ALARM
AND NOT   M00757	// R_2nd SS CLAMP.R UP/DN ALARM
AND NOT   M00758	// R_2nd SS CLAMP.L UP/DN ALARM
AND NOT   M00759	// R_2nd SS MANDREL BW/FW ALARM
AND NOT   M0075D	// R_2nd SS SPANKING BW/FW ALARM
AND NOT   M0076B	// R_2nd BD Z NOT MV
NOT
OR LOAD
LOAD NOT  M00680	// -
AND NOT   M00681	// -
AND NOT   M00682	// -
AND NOT   M00683	// -
AND NOT   M00684	// -
AND NOT   M00685	// -
AND NOT   M00686	// -
NOT
OR LOAD
LOAD NOT  M00760	// -
AND NOT   M00761	// -
AND NOT   M00762	// -
AND NOT   M00763	// -
AND NOT   M00764	// -
AND NOT   M00765	// -
AND NOT   M00766	// -
NOT
OR LOAD
LOAD NOT  M00770	// L_3rd BD Z NOT HOME
AND NOT   M00771	// L_1st CLP Z POS ERR
AND NOT   M00772	// L_3rd BD Z SVD ERR
AND NOT   M00773	// L_3rd BD Z NOT MV
AND NOT   M00774	// L_3rd BD Z +LIMIT
AND NOT   M00775	// L_1st CLP Z -LIMIT
AND NOT   M00776	// L_1st CLP Z NOT SERVO ON
NOT
OR LOAD
LOAD NOT  M00780	// R_3rd BD Z NOT HOME
AND NOT   M00781	// R_1st CLP Z POS ERR
AND NOT   M00782	// R_3rd BD Z SVD ERR
AND NOT   M00783	// R_3rd BD Z NOT MV
AND NOT   M00784	// R_3rd BD Z +LIMIT
AND NOT   M00785	// R_1st CLP Z -LIMIT
AND NOT   M00786	// R_1st CLP Z NOT SERVO ON
NOT
OR LOAD
MOVP      670 M0029
; L33
LOAD NOT  M00880
AND NOT   M00881
NOT
LOAD NOT  M00890
AND NOT   M00891
NOT
OR LOAD
MOVP      880 M0029
; L35
LOAD NOT  M00882
AND NOT   M00883
AND NOT   M00884	// L_4th SIDE ALIGN PRESSURE ALARM
NOT
LOAD NOT  M00892
AND NOT   M00893
AND NOT   M00894	// R_4th SIDE ALIGN PRESSURE ALARM
NOT
OR LOAD
MOVP      882 M0029
; L37
LOAD NOT  M00900	// IN BUFFER LEFT/RIGHT SN ALARM
AND NOT   M00901	// L_IN BUFFER VC ALARM
AND NOT   M00902	// OUT BUFFER LEFT/RIGHT SN ALARM
AND NOT   M00903	// L_OUT BUFFER VC ALARM
NOT
LOAD NOT  M00910
AND NOT   M00911	// R_IN BUFFER VC ALARM
AND NOT   M00912
AND NOT   M00913	// R_OUT BUFFER VC ALARM
NOT
OR LOAD
LOAD NOT  M0093A	// LF_2D CODE TM OUT
AND NOT   M0093B	// LF_2D CODE NG
AND NOT   M0093C	// RT_2D CODE TM OUT
AND NOT   M0093D	// RT_2D CODE NG
NOT
OR LOAD
MOVP      900 M0029
; L40
LOAD<>    0 M0092
MOVP      920 M0029
; L41
END

PROGRAM AUTO_LOAD (task: ½ºÄµ ÇÁ·Î±×·¥)

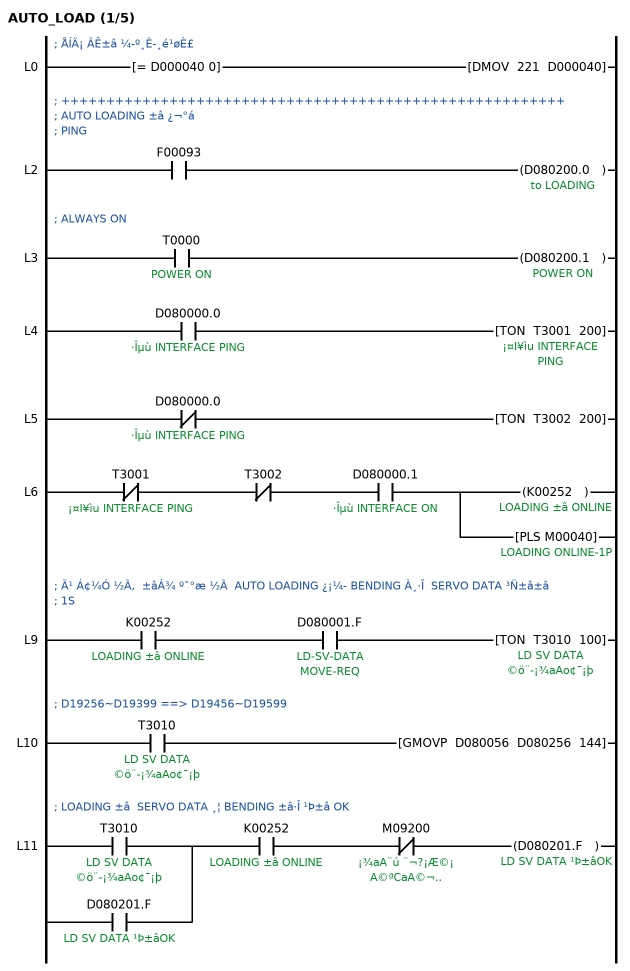
; L0
LOAD=     D000040 0
DMOV      221 D000040
// output comment: ÅÍÄ¡ ÃÊ±â ¼­º¸È­¸é¹øÈ£
// ++++++++++++++++++++++++++++++++++++++++++++++++++++++++
//    AUTO LOADING ±â ¿¬°á
; L2
LOAD      F00093
OUT       D080200.0	// to LOADING
// output comment: PING
; L3
LOAD      T0000	// POWER ON
OUT       D080200.1	// POWER ON
// output comment: ALWAYS ON
; L4
LOAD      D080000.0	// ·Îµù INTERFACE PING
TON       T3001 200	// ¡¤I¥ìu INTERFACE PING
; L5
LOAD NOT  D080000.0	// ·Îµù INTERFACE PING
TON       T3002 200
; L6
LOAD NOT  T3001	// ¡¤I¥ìu INTERFACE PING
AND NOT   T3002
AND       D080000.1	// ·Îµù INTERFACE ON
OUT       K00252	// LOADING ±â ONLINE
OUTP      M00040	// LOADING ONLINE-1P
// Ã¹ Á¢¼Ó ½Ã,  ±âÁ¾ º¯°æ ½Ã  AUTO LOADING ¿¡¼­ BENDING À¸·Î  SERVO DATA ³Ñ±â±â
; L9
LOAD      K00252	// LOADING ±â ONLINE
AND       D080001.F	// LD-SV-DATA MOVE-REQ
TON       T3010 100	// LD SV DATA ©ö¨­¡¾aAo¢¯¡þ
// output comment: 1S
; L10
LOAD      T3010	// LD SV DATA ©ö¨­¡¾aAo¢¯¡þ
GMOVP     D080056 D080256 144
// output comment: D19256~D19399 ==> D19456~D19599
; L11
LOAD      T3010	// LD SV DATA ©ö¨­¡¾aAo¢¯¡þ
OR        D080201.F	// LD SV DATA ¹Þ±âOK
AND       K00252	// LOADING ±â ONLINE
AND NOT   M09200	// ¡¾aA¨ú ¨¬?¡Æ©¡ A©ªCaA©¬..
OUT       D080201.F	// LD SV DATA ¹Þ±âOK
// output comment: LOADING ±â  SERVO DATA ¸¦ BENDING ±â·Î ¹Þ±â OK

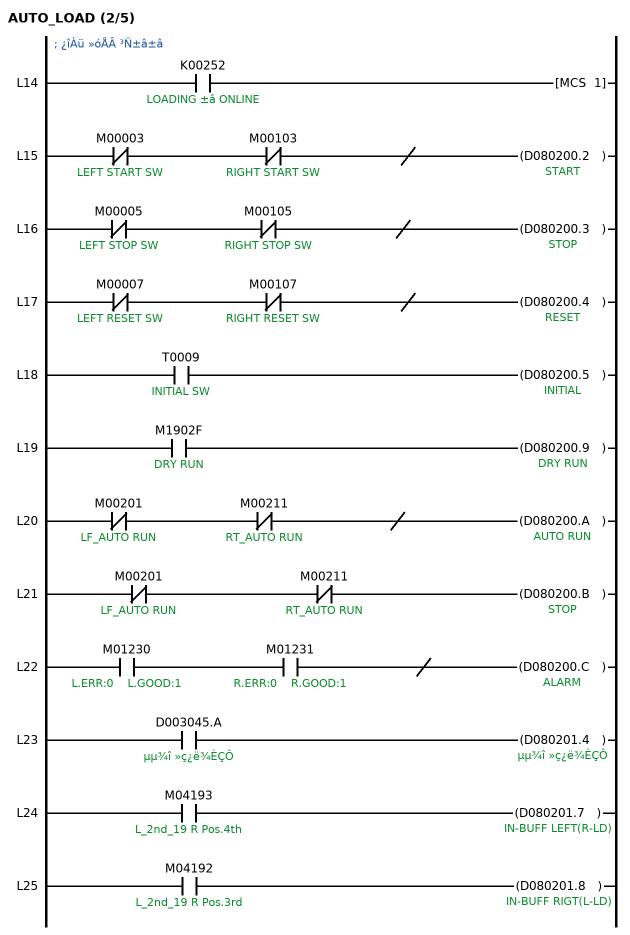
// ¿îÀü »óÅÂ ³Ñ±â±â
; L14
LOAD      K00252	// LOADING ±â ONLINE
MCS       1
; L15
LOAD NOT  M00003	// LEFT START SW
AND NOT   M00103	// RIGHT START SW
NOT
OUT       D080200.2	// START
; L16
LOAD NOT  M00005	// LEFT STOP SW
AND NOT   M00105	// RIGHT STOP SW
NOT
OUT       D080200.3	// STOP
; L17
LOAD NOT  M00007	// LEFT RESET SW
AND NOT   M00107	// RIGHT RESET SW
NOT
OUT       D080200.4	// RESET
; L18
LOAD      T0009	// INITIAL SW
OUT       D080200.5	// INITIAL
; L19
LOAD      M1902F	// DRY RUN
OUT       D080200.9	// DRY RUN
; L20
LOAD NOT  M00201	// LF_AUTO RUN
AND NOT   M00211	// RT_AUTO RUN
NOT
OUT       D080200.A	// AUTO RUN
; L21
LOAD NOT  M00201	// LF_AUTO RUN
AND NOT   M00211	// RT_AUTO RUN
OUT       D080200.B	// STOP
; L22
LOAD      M01230	// L.ERR:0    L.GOOD:1
AND       M01231	// R.ERR:0    R.GOOD:1
NOT
OUT       D080200.C	// ALARM
; L23
LOAD      D003045.A	// µµ¾î »ç¿ë¾ÈÇÔ
OUT       D080201.4	// µµ¾î »ç¿ë¾ÈÇÔ
; L24
LOAD      M04193	// L_2nd_19 R Pos.4th 
OUT       D080201.7	// IN-BUFF LEFT(R-LD)
; L25
LOAD      M04192	// L_2nd_19 R Pos.3rd
OUT       D080201.8	// IN-BUFF RIGT(L-LD)

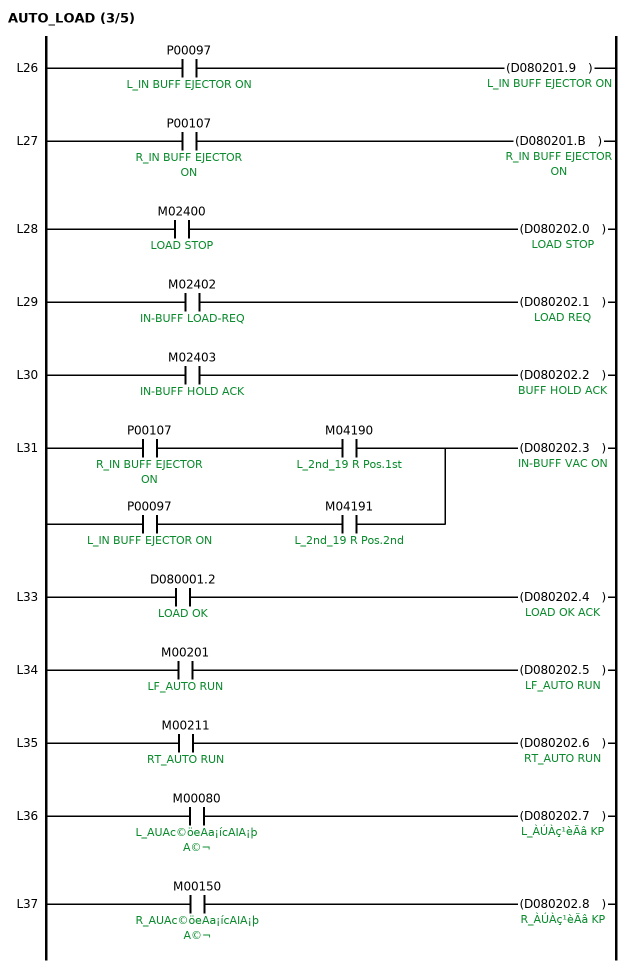
; L26
LOAD      P00097	// L_IN BUFF EJECTOR ON
OUT       D080201.9	// L_IN BUFF EJECTOR ON
; L27
LOAD      P00107	// R_IN BUFF EJECTOR ON
OUT       D080201.B	// R_IN BUFF EJECTOR ON
; L28
LOAD      M02400	// LOAD STOP
OUT       D080202.0	// LOAD STOP
; L29
LOAD      M02402	// IN-BUFF LOAD-REQ
OUT       D080202.1	// LOAD REQ
; L30
LOAD      M02403	// IN-BUFF HOLD ACK
OUT       D080202.2	// BUFF HOLD ACK
; L31
LOAD      P00107	// R_IN BUFF EJECTOR ON
AND       M04190	// L_2nd_19 R Pos.1st 
LOAD      P00097	// L_IN BUFF EJECTOR ON
AND       M04191	// L_2nd_19 R Pos.2nd
OR LOAD
OUT       D080202.3	// IN-BUFF VAC ON
; L33
LOAD      D080001.2	// LOAD OK
OUT       D080202.4	// LOAD OK ACK
; L34
LOAD      M00201	// LF_AUTO RUN
OUT       D080202.5	// LF_AUTO RUN
; L35
LOAD      M00211	// RT_AUTO RUN
OUT       D080202.6	// RT_AUTO RUN
; L36
LOAD      M00080	// L_AUAc©öeAa¡ícAIA¡þA©¬
OUT       D080202.7	// L_ÀÚÀç¹èÃâ KP
; L37
LOAD      M00150	// R_AUAc©öeAa¡ícAIA¡þA©¬
OUT       D080202.8	// R_ÀÚÀç¹èÃâ KP

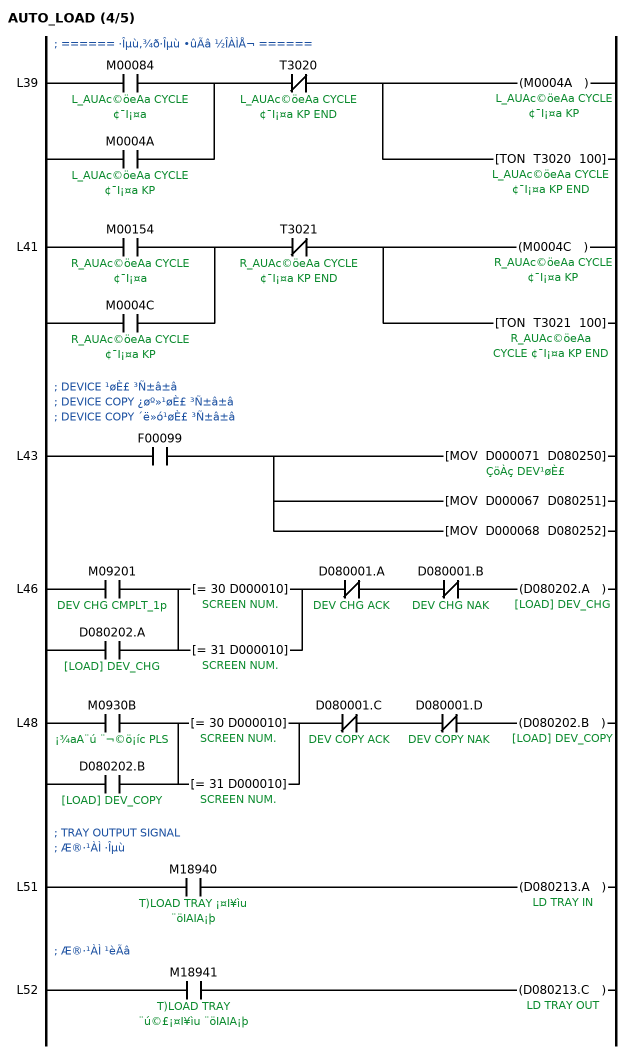
// ====== ·Îµù,¾ð·Îµù •ûÃâ ½ÎÀÌÅ¬ ======
; L39
LOAD      M00084	// L_AUAc©öeAa CYCLE ¢¯I¡¤a
OR        M0004A	// L_AUAc©öeAa CYCLE ¢¯I¡¤a KP
AND NOT   T3020	// L_AUAc©öeAa CYCLE ¢¯I¡¤a KP END
OUT       M0004A	// L_AUAc©öeAa CYCLE ¢¯I¡¤a KP
TON       T3020 100	// L_AUAc©öeAa CYCLE ¢¯I¡¤a KP END
; L41
LOAD      M00154	// R_AUAc©öeAa CYCLE ¢¯I¡¤a
OR        M0004C	// R_AUAc©öeAa CYCLE ¢¯I¡¤a KP
AND NOT   T3021	// R_AUAc©öeAa CYCLE ¢¯I¡¤a KP END
OUT       M0004C	// R_AUAc©öeAa CYCLE ¢¯I¡¤a KP
TON       T3021 100	// R_AUAc©öeAa CYCLE ¢¯I¡¤a KP END
; L43
LOAD      F00099
MOV       D000071 D080250	// ÇöÀç DEV¹øÈ£
MOV       D000067 D080251
MOV       D000068 D080252
// output comment: DEVICE ¹øÈ£ ³Ñ±â±â
// output comment: DEVICE COPY ¿øº»¹øÈ£ ³Ñ±â±â
// output comment: DEVICE COPY ´ë»ó¹øÈ£ ³Ñ±â±â
; L46
LOAD      M09201	// DEV CHG CMPLT_1p
OR        D080202.A	// [LOAD] DEV_CHG
LOAD=     30 D000010	// SCREEN NUM.
OR=       31 D000010	// SCREEN NUM.
AND LOAD
AND NOT   D080001.A	// DEV CHG ACK
AND NOT   D080001.B	// DEV CHG NAK
OUT       D080202.A	// [LOAD] DEV_CHG
; L48
LOAD      M0930B	// ¡¾aA¨ú ¨¬©ö¡íc PLS
OR        D080202.B	// [LOAD] DEV_COPY
LOAD=     30 D000010	// SCREEN NUM.
OR=       31 D000010	// SCREEN NUM.
AND LOAD
AND NOT   D080001.C	// DEV COPY ACK
AND NOT   D080001.D	// DEV COPY NAK
OUT       D080202.B	// [LOAD] DEV_COPY
// TRAY OUTPUT SIGNAL
; L51
LOAD      M18940	// T)LOAD TRAY ¡¤I¥ìu ¨öIAIA¡þ
OUT       D080213.A	// LD TRAY IN
// output comment: Æ®·¹ÀÌ ·Îµù
; L52
LOAD      M18941	// T)LOAD TRAY ¨ú©£¡¤I¥ìu ¨öIAIA¡þ
OUT       D080213.C	// LD TRAY OUT
// output comment: Æ®·¹ÀÌ ¹èÃâ

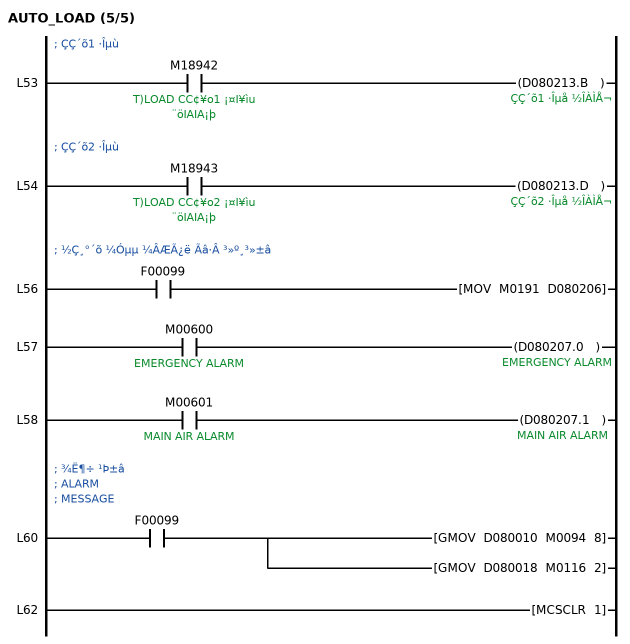
; L53
LOAD      M18942	// T)LOAD CC¢¥o1 ¡¤I¥ìu ¨öIAIA¡þ
OUT       D080213.B	// ÇÇ´õ1 ·Îµå ½ÎÀÌÅ¬
// output comment: ÇÇ´õ1 ·Îµù
; L54
LOAD      M18943	// T)LOAD CC¢¥o2 ¡¤I¥ìu ¨öIAIA¡þ
OUT       D080213.D	// ÇÇ´õ2 ·Îµå ½ÎÀÌÅ¬
// output comment: ÇÇ´õ2 ·Îµù
// ½Ç¸°´õ ¼Óµµ ¼ÂÆÃ¿ë Ãâ·Â ³»º¸³»±â
; L56
LOAD      F00099
MOV       M0191 D080206
; L57
LOAD      M00600	// EMERGENCY ALARM
OUT       D080207.0	// EMERGENCY ALARM
; L58
LOAD      M00601	// MAIN AIR ALARM
OUT       D080207.1	// MAIN AIR ALARM
// ¾Ë¶÷ ¹Þ±â
; L60
LOAD      F00099
GMOV      D080010 M0094 8
GMOV      D080018 M0116 2
// output comment: ALARM
// output comment: MESSAGE
; L62
MCSCLR    1

PROGRAM AUTO_UNLOAD (task: ½ºÄµ ÇÁ·Î±×·¥)

